// TwinCAT 3 PLC project PLC_HMI
// ProgramVersion: 3.1.4024.0
// libraries:
//   Tc2_DataExchange, * (Beckhoff Automation GmbH)
//   Tc2_Standard, * (Beckhoff Automation GmbH)
//   Tc2_System, * (Beckhoff Automation GmbH)
//   Tc2_Utilities, * (Beckhoff Automation GmbH)
//   Tc3_Database, * (Beckhoff Automation GmbH)
//   Tc3_EventLogger, * (Beckhoff Automation GmbH)
//   Tc3_Module, * (Beckhoff Automation GmbH)
// project tree:
//   DUTs/ ST_Alarm.TcDUT, ST_Error_Station_Handling.TcDUT, ST_Error_Description_Handling.TcDUT, ST_For_Screen.TcDUT, ST_For_Screen_New.TcDUT, ST_UserManagment.TcDUT
//   GVLs/ GVL_Error.TcGVL, GVL_Gauge.TcGVL, GVL_Recipe.TcGVL, GVL_USER.TcGVL, GVL_HIS.TcGVL, GVL_USER_UF.TcGVL, GVL_USER_UP.TcGVL
//   NotUsedPOU/ FB_AssignUserParam.TcPOU, F_ParseKeyValue.TcPOU, F_ParseUserString.TcPOU, F_SplitStringLines.TcPOU, P_EvtLog.TcPOU, P_ParseString.TcPOU, P_UserDataManagment.TcPOU
//   / PlcTask.TcTTO
//   POUs/ FB_Persistent.TcPOU, FB_SaveLineToFile.TcPOU, FB_SaveTextToFile.TcPOU, MAIN.TcPOU, P_ADS_ERR.TcPOU, P_ADS_Gauge.TcPOU, P_Error_Handling.TcPOU, P_Gauge_Measures.TcPOU, P_History_New.TcPOU, P_Recipebackup.TcPOU, P_ADS_1.TcPOU, P_History.TcPOU, P_Time.TcPOU, P_UserManagment.TcPOU, P_UserManagment_UP.TcPOU, P_UserManagment_UF.TcPOU
// real-time tasks:
//   TASK MainTask: cycle T#3ms, priority 20, ADS port 350
//   TASK SafetyTask: cycle T#10ms, priority 21, ADS port 351
//   TASK WeightTask: cycle T#1ms, priority 10, ADS port 352
//   TASK plctaskhmi: cycle T#10ms, priority 30, ADS port 353
//   TASK TaskToRefreshEAP: cycle T#8ms, priority 1, ADS port 301
//   TASK PlcTask: cycle T#10ms, priority 23, ADS port 354

CONFIGURATION PLC_HMI
    RESOURCE PLC ON TwinCAT3
        TASK PlcTask(INTERVAL := T#10ms, PRIORITY := 30);
        PROGRAM MAIN WITH PlcTask : MAIN;
    END_RESOURCE
END_CONFIGURATION

// ---- DUTs/ST_Alarm.TcDUT
TYPE ST_Alarm :
STRUCT
	sTekst1				: WSTRING(255);
	sTekst2				: WSTRING(255);
	sTekst3				: WSTRING(255);
	dtUtworzenia		: DT;
	iNumer				: INT;
	historical_alarm	: WSTRING(1000);
END_STRUCT
END_TYPE

// ---- DUTs/ST_Error_Station_Handling.TcDUT
TYPE ST_Error_Station_Handling :
STRUCT
	udiStationInError			:UDINT;
	wsStasionInError				:WSTRING(255);
END_STRUCT
END_TYPE

// ---- DUTs/ST_Error_Description_Handling.TcDUT
TYPE ST_Error_Description_Handling :
STRUCT
	udiStationErrorCode		:UDINT;
	wsStationErrorDescription	:WSTRING(255);	
END_STRUCT
END_TYPE

// ---- DUTs/ST_For_Screen.TcDUT
TYPE ST_For_Screen :
STRUCT
	data				:WSTRING(255);
	alarmy				:WSTRING(1000);
	user				:WSTRING(80);
	bErrorOccure		:BOOL := FALSE;
END_STRUCT
END_TYPE

// ---- DUTs/ST_For_Screen_New.TcDUT
TYPE ST_For_Screen_New :
STRUCT
	data				:WSTRING(255);
	alarmy				:WSTRING(1000);
	alarmy_id			:UDINT;
	stacja				:UDINT;
	user				:WSTRING(80);
	bErrorOccure		:BOOL := FALSE;
END_STRUCT
END_TYPE

// ---- DUTs/ST_UserManagment.TcDUT
TYPE ST_UserManagment :
STRUCT
	userID 				:	INT;			//numer porządkowy użytkownika
	domain				:	STRING(80);
	enabled				:	BOOL;
	userLogin			:	STRING(80);		//login do zalogowania
	userNameSurname 	:	WSTRING(255);	//imię i nazwisko
	userNameSurnameNumber	:UINT;
	password			:	STRING(255);	//hasło kalwiaturowe
	passwordRFID		:	STRING(255);	//hasło rfid
	passwordQR			:	STRING(255);	//hasło qr
	userGroup			:	STRING(80);		//grupa użytkowników
	userGropuNumber		:	UINT;			//numer grupy
	autoLogOff			:	STRING(80);		//czas do wylogowania
	locale				:	STRING(80);		//gdzie zapisujemy
	timeFormatlocale	:	STRING(80);		//format godziny
	timeZone			:	STRING(80);		//strefa czasowa
	signedPassword		:	STRING(80);		//hasło przekazywane do HMI
END_STRUCT
END_TYPE

// ---- GVLs/GVL_Error.TcGVL
{attribute 'qualified_only'}
VAR_GLOBAL PERSISTENT
	udi_Station_In_Error			:UDINT;
	udi_Station_In_Error_Code		:UDINT;
	ws_Stasion_In_Error				:WSTRING;
	ws_Station_Error_Description		:WSTRING(255);
	ws_Station_Error_Description_2	:WSTRING(255);
	A_Error_station	:ARRAY[0..100] OF ST_Error_Station_Handling; 
	A_Error_description	:ARRAY[0..500] OF ST_Error_Description_Handling;
	
	b_empy_error					:BOOL;
	b_new_system					:BOOL;
END_VAR
VAR_GLOBAL
	logowanie_krok: INT;
END_VAR

// ---- GVLs/GVL_Gauge.TcGVL
{attribute 'qualified_only'}
VAR_GLOBAL
	//input
	lr_WeightMass_recipe	:LREAL;
	lr_Dispencer1WeightMeasured	:LREAL;
	lr_Dispencer2WeightMeasured	:LREAL;
	lr_Dispencer3WeightMeasured	:LREAL;
	lr_Dispencer4WeightMeasured	:LREAL;
	lr_Tolerance_Low			:LREAL;
	lr_Tolerance_High			:LREAL;
	lr_weight_measured_1		:LREAL;
	lr_weight_measured_2		:LREAL;
	lr_weight_measured_3		:LREAL;
	lr_weight_measured_4		:LREAL;
	
	lr_mass_value_1				:LREAL;
	lr_mass_value_2				:LREAL;
	lr_mass_value_3				:LREAL;
	lr_mass_value_4				:LREAL;
	
	
	//output
	lr_out_max_weight_value :LREAL;
	lr_out_min_tolerance_low :LREAL;
	lr_out_max_tolerance_high :LREAL;
	
	lr_out_weight_measured_1 :LREAL;
	lr_out_weight_measured_2 :LREAL;
	lr_out_weight_measured_3 :LREAL;
	lr_out_weight_measured_4 :LREAL;
	
	s_actual_weight_1	:STRING;
	s_actual_weight_2	:STRING;	
	s_actual_weight_3	:STRING;
	s_actual_weight_4	:STRING;
	
	s_actual_weight_1_diff	:STRING;
	s_actual_weight_2_diff	:STRING;
	s_actual_weight_3_diff	:STRING;
	s_actual_weight_4_diff	:STRING;

	s_actual_corr_1		:STRING;
	s_actual_corr_2		:STRING;
	s_actual_corr_3		:STRING;
	s_actual_corr_4		:STRING;	
	
	s_actual_dose_1		:STRING;
	s_actual_dose_2		:STRING;
	s_actual_dose_3		:STRING;
	s_actual_dose_4		:STRING;
	
	lr_corr_add_1	:LREAL;
	lr_corr_sub_1	:LREAL;
	lr_corr_add_2	:LREAL;
	lr_corr_sub_2	:LREAL;
	lr_corr_add_3	:LREAL;
	lr_corr_sub_3	:LREAL;
	lr_corr_add_4	:LREAL;
	lr_corr_sub_4	:LREAL;
	
	s_actual_torque_1	:STRING;
	s_actual_torque_2	:STRING;
	s_actual_torque_diff_1		:STRING;
	s_actual_torque_diff_2		:STRING;
	
	s_actual_level_1	:STRING;
	s_actual_level_2	:STRING;
	
	lr_out_torque_low_1		:LREAL;
	lr_out_torque_low_2		:LREAL;
	lr_out_torque_high_1		:LREAL;
	lr_out_torque_high_2		:LREAL;	

	
END_VAR

// ---- GVLs/GVL_Recipe.TcGVL
{attribute 'qualified_only'}
VAR_GLOBAL
	b_recipe_backup	:BOOL;
END_VAR

// ---- GVLs/GVL_USER.TcGVL
{attribute 'qualified_only'}
VAR_GLOBAL PERSISTENT
		// wejścia cyfrowe
	user_array 					: ARRAY[1..100] OF ST_UserManagment;  // Tablica użytkowników
    currentUser 				: INT := 1;  // Indeks bieżącego użytkownika (zaczyna od 1)
    string_of_properties 		: STRING(1000);  // String z HMI z danymi użytkowników
	outside_accept_login		:BOOL;
	outside_login_pool			:STRING(255);  
	new_user_added				:BOOL;		//dodano użytkownika w PLC
	user_eddited				:BOOL; 		//zedytowano użytkownika w PLC
	b_new_users					:BOOL;		//wgranie uzytkowników
	currentUserName 			:WSTRING(255);
	currentUserGroup			:STRING(80);
	currentUserGroupNumber		:UINT;
	actualUserOn_UserName		:STRING(80);
	b_rewrite_main_users		:BOOL:=FALSE;
	
	logout						:BOOL;
	
	user_try_to_log				:BOOL;
	user_accept_to_log_in		:BOOL;
	no_user_found				:BOOL;
	user_succesed_log			:BOOL;
	putted_user_password		:STRING(255);  //pole w które użytkownik wpisuje hasło
	
	new_user					:BOOL;			//inicjalizacja dodawania nowego użytkownika
	new_user_accept				:BOOL;			//akceptacja dodania nowego użytkownika
	newuserNameSurname 			:WSTRING(255);	//imię i nazwisko
	newpassword					:STRING(255);	//hasło
	newpasswordRFID				:STRING(255);	//hasło rfid
	newpasswordQR				:STRING(255);	//hasło qr
	newuserGroup				:STRING(80);		//grupa użytkowników
	newuserGroupNumber			:UINT;
	newautoLogOff				:STRING(80);			//czas do wylogowania
	newlocale					:STRING(80);		//gdzie zapisujemy
	newtimeFormatlocale			:STRING(80);		//format godziny
	newtimeZone					:STRING(80);		//strefa czasowa
	
	edit_user					:BOOL;				//inicjalizacja edycji użytkownika
	edit_user_accept			:BOOL;			//akceptacja edycji użytkownika
	actual_editted_user			:WSTRING(255);	//wybór aktualnie edytowanego użytkownika
	edituserNameSurname 		:WSTRING(255);	//imię i nazwisko
	editpassword				:STRING(255);	//hasło
	editpasswordRFID			:STRING(255);	//hasło rfid
	editpasswordQR				:STRING(255);	//hasło qr
	edituserGroup				:STRING(80);	//grupa użytkowników
	editUserGroupNumber			:UINT;
	editautoLogOff				:STRING(80);	//czas do wylogowania
	edit_user_qr_or_rfid_password	:BOOL;		//edycja kodów rfid lub qr
		
	//wyjścia cyfrowe
	new_user_add_error			:BOOL;
	edit_user_error				:BOOL;
	bwait						:BOOL;
		
	delete_user						:BOOL;
	delete_user_accept				:BOOL;
	delete_user_error				:BOOL;
	choosen_to_delete				:WSTRING(255);
	user_deleted_succes				:BOOL;
	
	password_to_log_in				:STRING(80); //hasło do pola (1 z 5 (adm, opr, ser, tech, mech)
	
	b_rewrite_users_after_issues	:BOOL:=FALSE;
	
	b_user_drop_the_login			:BOOL;
	
	
	i_choosen_language :INT:=1;
END_VAR

// ---- GVLs/GVL_HIS.TcGVL
{attribute 'qualified_only'}
VAR_GLOBAL PERSISTENT
	// wyjścia cyfrowe
	Historical_array 			: ARRAY [1..1000] OF WSTRING(1000);
	ST_Alarmy 					: ARRAY [1..1000] OF st_for_screen;
	ST_Alarmy_ar1 				: ARRAY [0..28] OF st_for_screen;
	ST_Alarmy_New				:ARRAY  [1..1000] OF st_for_screen_new;
	ST_Alarmy_ar2 				: ARRAY [0..28] OF st_for_screen_new;
	user_for_alarms	 			: WSTRING(80);
	bclearhistory				: BOOL;
	s_time_mainscreen			: WSTRING(80);
	b_next_hist_page			:BOOL;
	b_prev_hist_page			:BOOL;
	i_start_index				:INT:=0;
END_VAR

// ---- GVLs/GVL_USER_UF.TcGVL
{attribute 'qualified_only'}
VAR_GLOBAL PERSISTENT
		// wejścia cyfrowe
	user_array 					: ARRAY[1..100] OF ST_UserManagment;  // Tablica użytkowników
    currentUser 				: INT := 1;  // Indeks bieżącego użytkownika (zaczyna od 1)
    string_of_properties 		: STRING(1000);  // String z HMI z danymi użytkowników
	outside_accept_login		:BOOL;
	outside_login_pool			:STRING(255);  
	new_user_added				:BOOL;		//dodano użytkownika w PLC
	user_eddited				:BOOL; 		//zedytowano użytkownika w PLC
	b_new_users					:BOOL;		//wgranie uzytkowników
	currentUserName 			:WSTRING(255);
	currentUserGroup			:STRING(80);
	actualUserOn_UserName		:STRING(80);
	b_rewrite_main_users		:BOOL:=FALSE;
	
	logout						:BOOL;
	
	user_try_to_log				:BOOL;
	user_accept_to_log_in		:BOOL;
	no_user_found				:BOOL;
	user_succesed_log			:BOOL;
	putted_user_password		:STRING(255);  //pole w które użytkownik wpisuje hasło
	
	new_user					:BOOL;			//inicjalizacja dodawania nowego użytkownika
	new_user_accept				:BOOL;			//akceptacja dodania nowego użytkownika
	newuserNameSurname 			:WSTRING(255);	//imię i nazwisko
	newpassword					:STRING(255);	//hasło
	newpasswordRFID				:STRING(255);	//hasło rfid
	newpasswordQR				:STRING(255);	//hasło qr
	newuserGroup				:STRING(80);		//grupa użytkowników
	newautoLogOff				:STRING(80);			//czas do wylogowania
	newlocale					:STRING(80);		//gdzie zapisujemy
	newtimeFormatlocale			:STRING(80);		//format godziny
	newtimeZone					:STRING(80);		//strefa czasowa
	
	edit_user					:BOOL;				//inicjalizacja edycji użytkownika
	edit_user_accept			:BOOL;			//akceptacja edycji użytkownika
	actual_editted_user			:WSTRING(255);	//wybór aktualnie edytowanego użytkownika
	edituserNameSurname 		:WSTRING(255);	//imię i nazwisko
	editpassword				:STRING(255);	//hasło
	editpasswordRFID			:STRING(255);	//hasło rfid
	editpasswordQR				:STRING(255);	//hasło qr
	edituserGroup				:STRING(80);		//grupa użytkowników
	editautoLogOff				:STRING(80);			//czas do wylogowania
	edit_user_qr_or_rfid_password	:BOOL;		//edycja kodów rfid lub qr
		
	//wyjścia cyfrowe
	new_user_add_error			:BOOL;
	edit_user_error				:BOOL;
	bwait						:BOOL;
		
	delete_user						:BOOL;
	delete_user_accept				:BOOL;
	delete_user_error				:BOOL;
	choosen_to_delete				:WSTRING(255);
	user_deleted_succes				:BOOL;
	
	password_to_log_in				:STRING(80); //hasło do pola (1 z 5 (adm, opr, ser, tech, mech)
	
	b_rewrite_users_after_issues	:BOOL:=FALSE;
	
	
END_VAR

// ---- GVLs/GVL_USER_UP.TcGVL
{attribute 'qualified_only'}
VAR_GLOBAL PERSISTENT
		// wejścia cyfrowe
	user_array 					: ARRAY[1..100] OF ST_UserManagment;  // Tablica użytkowników
    currentUser 				: INT := 1;  // Indeks bieżącego użytkownika (zaczyna od 1)
    string_of_properties 		: STRING(1000);  // String z HMI z danymi użytkowników
	outside_accept_login		:BOOL;
	outside_login_pool			:STRING(255);  
	new_user_added				:BOOL;		//dodano użytkownika w PLC
	user_eddited				:BOOL; 		//zedytowano użytkownika w PLC
	b_new_users					:BOOL;		//wgranie uzytkowników
	currentUserName 			:WSTRING(255);
	currentUserGroup			:STRING(80);
	actualUserOn_UserName		:STRING(80);
	b_rewrite_main_users		:BOOL:=FALSE;
	
	logout						:BOOL;
	
	user_try_to_log				:BOOL;
	user_accept_to_log_in		:BOOL;
	no_user_found				:BOOL;
	user_succesed_log			:BOOL;
	putted_user_password		:STRING(255);  //pole w które użytkownik wpisuje hasło
	
	new_user					:BOOL;			//inicjalizacja dodawania nowego użytkownika
	new_user_accept				:BOOL;			//akceptacja dodania nowego użytkownika
	newuserNameSurname 			:WSTRING(255);	//imię i nazwisko
	newpassword					:STRING(255);	//hasło
	newpasswordRFID				:STRING(255);	//hasło rfid
	newpasswordQR				:STRING(255);	//hasło qr
	newuserGroup				:STRING(80);		//grupa użytkowników
	newautoLogOff				:STRING(80);			//czas do wylogowania
	newlocale					:STRING(80);		//gdzie zapisujemy
	newtimeFormatlocale			:STRING(80);		//format godziny
	newtimeZone					:STRING(80);		//strefa czasowa
	
	edit_user					:BOOL;				//inicjalizacja edycji użytkownika
	edit_user_accept			:BOOL;			//akceptacja edycji użytkownika
	actual_editted_user			:WSTRING(255);	//wybór aktualnie edytowanego użytkownika
	edituserNameSurname 		:WSTRING(255);	//imię i nazwisko
	editpassword				:STRING(255);	//hasło
	editpasswordRFID			:STRING(255);	//hasło rfid
	editpasswordQR				:STRING(255);	//hasło qr
	edituserGroup				:STRING(80);		//grupa użytkowników
	editautoLogOff				:STRING(80);			//czas do wylogowania
	edit_user_qr_or_rfid_password	:BOOL;		//edycja kodów rfid lub qr
		
	//wyjścia cyfrowe
	new_user_add_error			:BOOL;
	edit_user_error				:BOOL;
	bwait						:BOOL;
		
	delete_user						:BOOL;
	delete_user_accept				:BOOL;
	delete_user_error				:BOOL;
	choosen_to_delete				:WSTRING(255);
	user_deleted_succes				:BOOL;
	
	password_to_log_in				:STRING(80); //hasło do pola (1 z 5 (adm, opr, ser, tech, mech)
	
	b_rewrite_users_after_issues	:BOOL:=FALSE;
	
	
END_VAR

// ---- POUs/MAIN.TcPOU
PROGRAM MAIN
VAR
		
END_VAR

P_ADS_1();
P_Time();
P_History();
P_History_New();
P_UserManagment();
P_Recipebackup();
P_Gauge_Measures();
P_ADS_Gauge();
P_ADS_Err();
P_Error_Handling();

END_PROGRAM

// ---- POUs/P_ADS_1.TcPOU
PROGRAM P_ADS_1
VAR
	sTextAlarm1				: WSTRING(255);
	sTextAlarm2				: WSTRING(255);
	sTextAlarm3				: WSTRING(255);
	user					: WSTRING(80);
	iNumberAlarm			: INT;
	bTrigger				: BOOL;
	
	fbRead_1: FB_ReadAdsSymByName;
	fbRead_2: FB_ReadAdsSymByName;
	fbRead_3: FB_ReadAdsSymByName;
	fbCyclicReadout: TON;
	fbRead_4: FB_ReadAdsSymByName;
	fbRead_5: FB_ReadAdsSymByName;
	fbLocaltime: FB_LocalSystemTime;

END_VAR

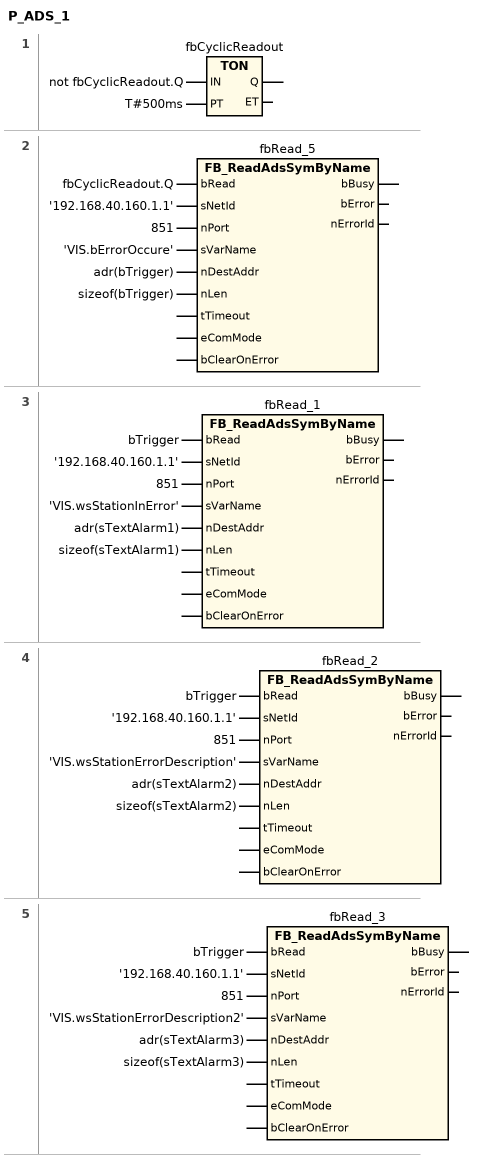
// NETWORK 1
fbCyclicReadout(IN := not fbCyclicReadout.Q, PT := T#500ms); // TON

// NETWORK 2
fbRead_5(
    bRead := fbCyclicReadout.Q,
    sNetId := '192.168.40.160.1.1',
    nPort := 851,
    sVarName := 'VIS.bErrorOccure',
    nDestAddr := adr(bTrigger),
    nLen := sizeof(bTrigger)); // FB_ReadAdsSymByName

// NETWORK 3
fbRead_1(
    bRead := bTrigger,
    sNetId := '192.168.40.160.1.1',
    nPort := 851,
    sVarName := 'VIS.wsStationInError',
    nDestAddr := adr(sTextAlarm1),
    nLen := sizeof(sTextAlarm1)); // FB_ReadAdsSymByName

// NETWORK 4
fbRead_2(
    bRead := bTrigger,
    sNetId := '192.168.40.160.1.1',
    nPort := 851,
    sVarName := 'VIS.wsStationErrorDescription',
    nDestAddr := adr(sTextAlarm2),
    nLen := sizeof(sTextAlarm2)); // FB_ReadAdsSymByName

// NETWORK 5
fbRead_3(
    bRead := bTrigger,
    sNetId := '192.168.40.160.1.1',
    nPort := 851,
    sVarName := 'VIS.wsStationErrorDescription2',
    nDestAddr := adr(sTextAlarm3),
    nLen := sizeof(sTextAlarm3)); // FB_ReadAdsSymByName

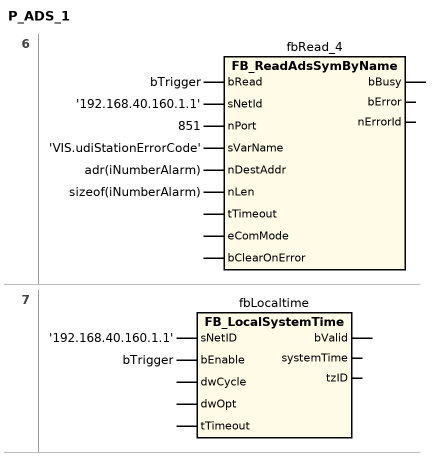
// NETWORK 6
fbRead_4(
    bRead := bTrigger,
    sNetId := '192.168.40.160.1.1',
    nPort := 851,
    sVarName := 'VIS.udiStationErrorCode',
    nDestAddr := adr(iNumberAlarm),
    nLen := sizeof(iNumberAlarm)); // FB_ReadAdsSymByName

// NETWORK 7
fbLocaltime(sNetID := '192.168.40.160.1.1', bEnable := bTrigger); // FB_LocalSystemTime

END_PROGRAM

// ---- POUs/P_Time.TcPOU
PROGRAM P_Time
VAR
    fbSystemTime : GETSYSTEMTIME;
    timeAsFileTime : T_FILETIME;
    timeAsDT : DT;
	actual_date_meawhile :DT;
	s_time_mainscreen	:WSTRING(80);
END_VAR


fbSystemTime(
    timeLoDW => timeAsFileTime.dwLowDateTime,
    timeHiDW => timeAsFileTime.dwHighDateTime 
);
timeAsDT := FILETIME_TO_DT(timeAsFileTime);
actual_date_meawhile:=timeAsDT;
actual_date_meawhile := actual_date_meawhile + T#2H;
s_time_mainscreen := DT_TO_WSTRING(actual_date_meawhile);
s_time_mainscreen := WRIGHT(s_time_mainscreen, WLEN(s_time_mainscreen) - 3);
gvl_his.s_time_mainscreen:=s_time_mainscreen;

END_PROGRAM

// ---- POUs/P_History.TcPOU
PROGRAM P_History
VAR
	nowyAlarm			: BOOL;
	i,j,k,n 			: INT; 
	m					: INT:=0;
	trescAlarmu1		: WSTRING(255);
	trescAlarmu2		: WSTRING(255);
	trescAlarmu3		: WSTRING(255);
	numerAlarmu			: INT;
	aktualnaData		: DT;
	
	bTrigerZapisu 		: R_TRIG;
	
	historical_alarm	: WSTRING(1000);
	tempDateString		: WSTRING(255);
	
	previousTrescAlarmu1 : WSTRING(255);
    previousTrescAlarmu2 : WSTRING(255);
    previousTrescAlarmu3 : WSTRING(255);
    previousNumerAlarmu  : INT;
    previousAktualnaData : DT;
	
	isAlarmChanged : BOOL := FALSE;
	
	isDuplicate: BOOL;
	bCzyszczenie :BOOL :=gvl_his.bclearhistory;
	bDuplikat :	BOOL;
	
	fbPersistent	: FB_Persistent;
	i_start_index		:INT;
	b_next_hist_page_old	:BOOL;
	b_prev_hist_page_old	:BOOL;
END_VAR

fbPersistent(
    bWrite := , 
    tInterval := T#30M, 
    bBusy => , 
    bErr => , 
    udErrID => 
);

trescAlarmu1 := P_ADS_1.sTextAlarm1;
trescAlarmu2 := P_ADS_1.sTextAlarm2;
trescAlarmu3 := P_ADS_1.sTextAlarm3;
numerAlarmu := P_ADS_1.iNumberAlarm;
aktualnaData := P_time.timeAsDT;

isAlarmChanged := (previousTrescAlarmu1 <> trescAlarmu1) OR
                  (previousTrescAlarmu2 <> trescAlarmu2) OR
                  (previousTrescAlarmu3 <> trescAlarmu3) OR
                  (previousNumerAlarmu <> numerAlarmu);

bTrigerZapisu(CLK := P_ADS_1.bTrigger);

IF bTrigerZapisu.Q OR isAlarmChanged THEN
    // Przesuwanie alarmów
    FOR i := 1000 TO 2 BY -1 DO
        GVL_HIS.Historical_array[i] := GVL_HIS.Historical_array[i - 1];
//		GVL_HIS.ST_Alarmy[i] := GVL_HIS.ST_Alarmy[i - 1];
     	GVL_HIS.ST_Alarmy[i].alarmy := GVL_HIS.ST_Alarmy[i - 1].alarmy;  // Przesunięcie struktury do przodu
		GVL_HIS.ST_Alarmy[i].data := GVL_HIS.ST_Alarmy[i - 1].data;
		GVL_HIS.ST_Alarmy[i].user := GVL_HIS.ST_Alarmy[i - 1].user;
		GVL_HIS.ST_Alarmy[i].bErrorOccure := GVL_HIS.ST_Alarmy[i - 1].bErrorOccure;
    END_FOR
    historical_alarm := WCONCAT(UDINT_TO_WSTRING(numerAlarmu), " | ");
    historical_alarm := WCONCAT(historical_alarm, trescAlarmu1);
    historical_alarm := WCONCAT(historical_alarm, " | ");
    historical_alarm := WCONCAT(historical_alarm, trescAlarmu2);
    historical_alarm := WCONCAT(historical_alarm, " | ");
    historical_alarm := WCONCAT(historical_alarm, trescAlarmu3);
    historical_alarm := WCONCAT(historical_alarm, " ");
    aktualnaData := aktualnaData + T#1H;
    tempDateString := DT_TO_WSTRING(aktualnaData);
    tempDateString := WRIGHT(tempDateString, WLEN(tempDateString) - 3);
//	historical_alarm := CONCAT(historical_alarm,tempDateString);

    IF WLEN(historical_alarm) >= 30 THEN
		
        GVL_HIS.Historical_array[1] := historical_alarm;     
		GVL_HIS.ST_Alarmy[1].alarmy := historical_alarm;      
        GVL_HIS.ST_Alarmy[1].data := tempDateString;         
        GVL_HIS.ST_Alarmy[1].user := gvl_his.user_for_alarms;         
        GVL_HIS.ST_Alarmy[1].bErrorOccure := TRUE;
        
        j := 1;
	
        FOR i := 1 TO 1000 DO
            IF WLEN(GVL_HIS.Historical_array[i]) >= 30 THEN
                GVL_HIS.Historical_array[j] := GVL_HIS.Historical_array[i];
				GVL_HIS.ST_Alarmy[j].alarmy := GVL_HIS.ST_Alarmy[i].alarmy; 
				GVL_HIS.ST_Alarmy[j].data := GVL_HIS.ST_Alarmy[i].data;
				GVL_HIS.ST_Alarmy[j].user := GVL_HIS.ST_Alarmy[i].user;
				GVL_HIS.ST_Alarmy[i].bErrorOccure := GVL_HIS.ST_Alarmy[i].bErrorOccure;
                j := j + 1;
            END_IF
        END_FOR

		IF j >= 500 THEN
            FOR i := 500 TO 1000 DO
                GVL_HIS.Historical_array[i] := "";  // Czyszczenie najstarszych wpisów
                GVL_HIS.ST_Alarmy[i].alarmy := "";  // Czyszczenie najstarszych alarmów
                GVL_HIS.ST_Alarmy[i].data := "";  
                GVL_HIS.ST_Alarmy[i].user := "";  
                GVL_HIS.ST_Alarmy[i].bErrorOccure := FALSE;
            END_FOR
            j := 500;  // Aktualizacja j, aby tablica miała maksymalnie 850 alarmów
        END_IF		

        FOR i := j TO 1000 DO
            GVL_HIS.Historical_array[i] := "";
			GVL_HIS.ST_Alarmy[i].alarmy := "";     
       		GVL_HIS.ST_Alarmy[i].data := "";           
      		GVL_HIS.ST_Alarmy[i].user := "";           
      		GVL_HIS.ST_Alarmy[i].bErrorOccure := FALSE;              
        END_FOR		
    END_IF
    
    previousTrescAlarmu1 := trescAlarmu1;
    previousTrescAlarmu2 := trescAlarmu2;
    previousTrescAlarmu3 := trescAlarmu3;
    previousNumerAlarmu := numerAlarmu;
	
	FOR i := 1000 TO 2 BY -1 DO
    isDuplicate := (GVL_HIS.ST_Alarmy[i].alarmy = GVL_HIS.ST_Alarmy[i-1].alarmy) AND
                   (GVL_HIS.ST_Alarmy[i].data = GVL_HIS.ST_Alarmy[i-1].data) AND
                   (GVL_HIS.ST_Alarmy[i].user = GVL_HIS.ST_Alarmy[i-1].user);
    	IF isDuplicate AND bDuplikat THEN
        		FOR j := i TO 1000 - 1 DO
            		GVL_HIS.ST_Alarmy[j] := GVL_HIS.ST_Alarmy[j + 1];
        		END_FOR
        	GVL_HIS.ST_Alarmy[1000].alarmy := "";
        	GVL_HIS.ST_Alarmy[1000].data := "";
        	GVL_HIS.ST_Alarmy[1000].user := "";
    	END_IF
	END_FOR

	IF bCzyszczenie THEN
		FOR i := 1 TO 1000 DO
    		GVL_HIS.ST_Alarmy[i].alarmy := ""; 
    		GVL_HIS.ST_Alarmy[i].data := "";   
    		GVL_HIS.ST_Alarmy[i].user := "";
			GVL_HIS.ST_Alarmy[i].bErrorOccure:=FALSE;    
		END_FOR
	END_IF
END_IF

IF gvl_his.b_next_hist_page = TRUE AND b_next_hist_page_old = FALSE AND gvl_his.i_start_index<20 THEN
	gvl_his.i_start_index:=gvl_his.i_start_index+1;
END_IF

IF gvl_his.b_prev_hist_page = TRUE AND b_prev_hist_page_old = FALSE AND gvl_his.i_start_index>0 THEN
	gvl_his.i_start_index:=gvl_his.i_start_index-1;
END_IF

b_next_hist_page_old := gvl_his.b_next_hist_page;
b_prev_hist_page_old := gvl_his.b_prev_hist_page;

i_start_index := gvl_his.i_start_index * 28;


IF (i_start_index > 0) AND (i_start_index<580) THEN
FOR m := 0 TO 28 DO
        gvl_his.ST_Alarmy_ar1[m].alarmy := gvl_his.ST_Alarmy[i_start_index + m].alarmy;
        gvl_his.ST_Alarmy_ar1[m].bErrorOccure := gvl_his.ST_Alarmy[i_start_index + m].bErrorOccure;
        gvl_his.ST_Alarmy_ar1[m].data := gvl_his.ST_Alarmy[i_start_index + m].data;
        gvl_his.ST_Alarmy_ar1[m].user := gvl_his.ST_Alarmy[i_start_index + m].user;
    END_FOR;
END_IF
IF i_start_index=0 THEN
		FOR m := 1 TO 28 DO
        gvl_his.ST_Alarmy_ar1[m].alarmy := gvl_his.ST_Alarmy[i_start_index + m].alarmy;
        gvl_his.ST_Alarmy_ar1[m].bErrorOccure := gvl_his.ST_Alarmy[i_start_index + m].bErrorOccure;
        gvl_his.ST_Alarmy_ar1[m].data := gvl_his.ST_Alarmy[i_start_index + m].data;
        gvl_his.ST_Alarmy_ar1[m].user := gvl_his.ST_Alarmy[i_start_index + m].user;
    	END_FOR;
END_IF;

END_PROGRAM

// ---- POUs/FB_Persistent.TcPOU
FUNCTION_BLOCK FB_Persistent

(********************************************************************************************************)
(*								Beckhoff Automation Poland												*)
(* 									FB_Persistent 	v1.5												*)
(* 										20.08.2014														*)
(* 							v1.5 - zmiana minimalnego interwalu zapisu									*)
(* 					Blok funkcyjny zapisujący zmienne typu persistent na karcie CF						*)
(* 						Możliwy zapis na żądanie lub z określoną częstotliwością.  						*)
(* 				Pozostawienie wejscia tInterval bez zmiennej wyłacza funkcję zapisu cyklicznego			*)
(* 							Minimalny czas między zapisem cyklicznym 30s								*)
(* 				Konieczne jest dodanie biblioteki TcUtilities.lib, TcSystem.lib oraz TcBase.lib			*)
(*			 UWAGA: Blok przygotowany dla RunTime 1 port 851 - typowa konfiguracja 						*)
(*______________________________________________________________________________________________________*)

VAR_INPUT
	bWrite					: BOOL;						(*Zapis na rozkaz *)
	tInterval				: TIME:=T#71582M47S295MS;	(*Czestotliwosc zapisu na karte CF*)
END_VAR
VAR_OUTPUT
	bBusy					: BOOL;
	bErr					: BOOL;
	udErrID					: UDINT;
END_VAR
VAR
	fbWritePersistentData	: FB_WritePersistentData; 	(* Blok zapisu *)
	t1						: TON;						(* Timer zapisu *)
	_GETCURTASKINDEX		: GETCURTASKINDEX;			(* Informacja o Tasku *)
	BIndex					: BYTE;						(* Nr tasku *)
END_VAR

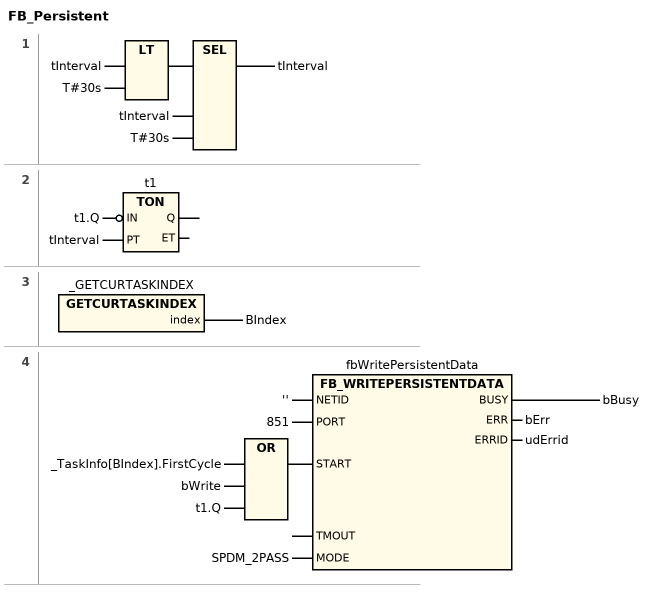
// NETWORK 1
tInterval := SEL(tInterval < T#30s, tInterval, T#30s);

// NETWORK 2
t1(IN := NOT t1.Q, PT := tInterval); // TON

// NETWORK 3
_GETCURTASKINDEX(); // GETCURTASKINDEX
BIndex := _GETCURTASKINDEX.index;

// NETWORK 4
fbWritePersistentData(
    NETID := '',
    PORT := 851,
    START := _TaskInfo[BIndex].FirstCycle OR bWrite OR t1.Q,
    MODE := SPDM_2PASS,
    ERR => bErr,
    ERRID => udErrid); // FB_WRITEPERSISTENTDATA
bBusy := fbWritePersistentData.BUSY;

END_FUNCTION_BLOCK

// ---- POUs/P_History_New.TcPOU
PROGRAM P_History_New
VAR
	nowyAlarm			: BOOL;
	i,j,k,n 			: INT; 
	m					: INT:=0;
	trescAlarmu1		: WSTRING(255);
	trescAlarmu2		: WSTRING(255);
	trescAlarmu3		: WSTRING(255);
	numerAlarmu			: INT;
	aktualnaData		: DT;
	station_id			:UDINT;
	alarm_id			:UDINT;
	
	bTrigerZapisu 		: R_TRIG;
	
	historical_alarm	: WSTRING(1000);
	historical_alarm_id	: UDINT;
	historical_station_id	:UDINT;
	tempDateString		: WSTRING(255);
	
	previousTrescAlarmu1 : WSTRING(255);
    previousTrescAlarmu2 : WSTRING(255);
    previousTrescAlarmu3 : WSTRING(255);
    previousNumerAlarmu  : INT;
    previousAktualnaData : DT;
	
	isAlarmChanged : BOOL := FALSE;
	
	isDuplicate: BOOL;
	bCzyszczenie :BOOL :=gvl_his.bclearhistory;
	bDuplikat :	BOOL;
	
	fbPersistent	: FB_Persistent;
	i_start_index		:INT;
	b_next_hist_page_old	:BOOL;
	b_prev_hist_page_old	:BOOL;
END_VAR

fbPersistent(
    bWrite := , 
    tInterval := T#30M, 
    bBusy => , 
    bErr => , 
    udErrID => 
);

trescAlarmu1 := P_ADS_1.sTextAlarm1;
trescAlarmu2 := P_ADS_1.sTextAlarm2;
trescAlarmu3 := P_ADS_1.sTextAlarm3;
numerAlarmu := P_ADS_1.iNumberAlarm;
aktualnaData := P_time.timeAsDT;
station_id	:=p_ads_err.udiStationInError;
alarm_id	:=p_ads_err.udiStationErrorCode;


isAlarmChanged := (previousTrescAlarmu1 <> trescAlarmu1) OR
                  (previousTrescAlarmu2 <> trescAlarmu2) OR
                  (previousTrescAlarmu3 <> trescAlarmu3) OR
                  (previousNumerAlarmu <> numerAlarmu);

bTrigerZapisu(CLK := P_ADS_1.bTrigger);

IF bTrigerZapisu.Q OR isAlarmChanged THEN
    // Przesuwanie alarmów
    FOR i := 1000 TO 2 BY -1 DO
        GVL_HIS.Historical_array[i] := GVL_HIS.Historical_array[i - 1];
//		GVL_HIS.ST_Alarmy[i] := GVL_HIS.ST_Alarmy[i - 1];
     	GVL_HIS.ST_Alarmy_New[i].alarmy := GVL_HIS.ST_Alarmy_New[i - 1].alarmy;  // Przesunięcie struktury do przodu
		GVL_HIS.ST_Alarmy_New[i].data := GVL_HIS.ST_Alarmy_New[i - 1].data;
		GVL_HIS.ST_Alarmy_New[i].user := GVL_HIS.ST_Alarmy_New[i - 1].user;
		GVL_HIS.ST_Alarmy_New[i].bErrorOccure := GVL_HIS.ST_Alarmy_New[i - 1].bErrorOccure;
		gvl_his.ST_Alarmy_New[i].alarmy_id:=gvl_his.ST_Alarmy_New[i-1].alarmy_id;
		gvl_his.ST_Alarmy_New[i].stacja:=gvl_his.ST_Alarmy_New[i-1].stacja;
    END_FOR
    historical_alarm := WCONCAT(UDINT_TO_WSTRING(numerAlarmu), " | ");
    historical_alarm := WCONCAT(historical_alarm, trescAlarmu1);
    historical_alarm := WCONCAT(historical_alarm, " | ");
    historical_alarm := WCONCAT(historical_alarm, trescAlarmu2);
    historical_alarm := WCONCAT(historical_alarm, " | ");
    historical_alarm := WCONCAT(historical_alarm, trescAlarmu3);
    historical_alarm := WCONCAT(historical_alarm, " ");
    aktualnaData := aktualnaData + T#1H;
    tempDateString := DT_TO_WSTRING(aktualnaData);
    tempDateString := WRIGHT(tempDateString, WLEN(tempDateString) - 3);
	historical_alarm_id:=alarm_id;
	historical_station_id:=station_id;
	
	
	
//	historical_alarm := CONCAT(historical_alarm,tempDateString);

    IF WLEN(historical_alarm) >= 30 THEN
		
        GVL_HIS.Historical_array[1] := historical_alarm;     
		GVL_HIS.ST_Alarmy_new[1].alarmy := historical_alarm;      
        GVL_HIS.ST_Alarmy_new[1].data := tempDateString;         
        GVL_HIS.ST_Alarmy_new[1].user := gvl_his.user_for_alarms;
		GVL_HIS.ST_Alarmy_new[1].alarmy_id:=historical_alarm_id;
		GVL_HIS.ST_Alarmy_new[1].stacja:=historical_station_id;         
        GVL_HIS.ST_Alarmy_new[1].bErrorOccure := TRUE;
        
        j := 1;
	
        FOR i := 1 TO 1000 DO
            IF WLEN(GVL_HIS.Historical_array[i]) >= 30 THEN
                GVL_HIS.Historical_array[j] := GVL_HIS.Historical_array[i];
				GVL_HIS.ST_Alarmy_new[j].alarmy := GVL_HIS.ST_Alarmy_new[i].alarmy; 
				GVL_HIS.ST_Alarmy_new[j].data := GVL_HIS.ST_Alarmy_new[i].data;
				GVL_HIS.ST_Alarmy_new[j].user := GVL_HIS.ST_Alarmy_new[i].user;
				GVL_HIS.ST_Alarmy_new[j].alarmy_id:=GVL_HIS.ST_Alarmy_new[i].alarmy_id;
				GVL_HIS.ST_Alarmy_new[j].stacja:=GVL_HIS.ST_Alarmy_new[i].stacja; 
				GVL_HIS.ST_Alarmy_new[j].bErrorOccure := GVL_HIS.ST_Alarmy_new[i].bErrorOccure;
                j := j + 1;
            END_IF
        END_FOR

		IF j >= 500 THEN
            FOR i := 500 TO 1000 DO
                GVL_HIS.Historical_array[i] := "";  // Czyszczenie najstarszych wpisów
                GVL_HIS.ST_Alarmy_new[i].alarmy := "";  // Czyszczenie najstarszych alarmów
                GVL_HIS.ST_Alarmy_new[i].data := "";  
                GVL_HIS.ST_Alarmy_new[i].user := "";
				GVL_HIS.ST_Alarmy_new[i].alarmy_id:=0;
				GVL_HIS.ST_Alarmy_new[i].stacja:=0;  
                GVL_HIS.ST_Alarmy_new[i].bErrorOccure := FALSE;
            END_FOR
            j := 500;  // Aktualizacja j, aby tablica miała maksymalnie 850 alarmów
        END_IF		

        FOR i := j TO 1000 DO
            GVL_HIS.Historical_array[i] := "";
			GVL_HIS.ST_Alarmy_new[i].alarmy := "";     
       		GVL_HIS.ST_Alarmy_new[i].data := "";           
      		GVL_HIS.ST_Alarmy_new[i].user := "";           
      		GVL_HIS.ST_Alarmy_new[i].bErrorOccure := FALSE;
			GVL_HIS.ST_Alarmy_new[i].alarmy_id:=0;
			GVL_HIS.ST_Alarmy_new[i].stacja:=0;               
        END_FOR		
    END_IF
    
    previousTrescAlarmu1 := trescAlarmu1;
    previousTrescAlarmu2 := trescAlarmu2;
    previousTrescAlarmu3 := trescAlarmu3;
    previousNumerAlarmu := numerAlarmu;
	
	FOR i := 1000 TO 2 BY -1 DO
    isDuplicate := (GVL_HIS.ST_Alarmy_new[i].alarmy = GVL_HIS.ST_Alarmy_new[i-1].alarmy) AND
                   (GVL_HIS.ST_Alarmy_new[i].data = GVL_HIS.ST_Alarmy_new[i-1].data) AND
                   (GVL_HIS.ST_Alarmy_new[i].user = GVL_HIS.ST_Alarmy_new[i-1].user);
    	IF isDuplicate AND bDuplikat THEN
        		FOR j := i TO 1000 - 1 DO
            		GVL_HIS.ST_Alarmy_new[j] := GVL_HIS.ST_Alarmy_new[j + 1];
        		END_FOR
        	GVL_HIS.ST_Alarmy_new[1000].alarmy := "";
        	GVL_HIS.ST_Alarmy_new[1000].data := "";
        	GVL_HIS.ST_Alarmy_new[1000].user := "";
			GVL_HIS.ST_Alarmy_new[1000].alarmy_id:=0;
			GVL_HIS.ST_Alarmy_new[1000].stacja:=0;   
    	END_IF
	END_FOR

	IF bCzyszczenie THEN
		FOR i := 1 TO 1000 DO
    		GVL_HIS.ST_Alarmy_new[i].alarmy := ""; 
    		GVL_HIS.ST_Alarmy_new[i].data := "";   
    		GVL_HIS.ST_Alarmy_new[i].user := "";
			GVL_HIS.ST_Alarmy_new[i].bErrorOccure:=FALSE;
			GVL_HIS.ST_Alarmy_new[i].alarmy_id:=0;
	        GVL_HIS.ST_Alarmy_new[i].stacja:=0;   
		END_FOR
	END_IF
END_IF

IF gvl_his.b_next_hist_page = TRUE AND b_next_hist_page_old = FALSE AND gvl_his.i_start_index<20 THEN
	gvl_his.i_start_index:=gvl_his.i_start_index+1;
END_IF

IF gvl_his.b_prev_hist_page = TRUE AND b_prev_hist_page_old = FALSE AND gvl_his.i_start_index>0 THEN
	gvl_his.i_start_index:=gvl_his.i_start_index-1;
END_IF

b_next_hist_page_old := gvl_his.b_next_hist_page;
b_prev_hist_page_old := gvl_his.b_prev_hist_page;

i_start_index := gvl_his.i_start_index * 28;


IF (i_start_index > 0) AND (i_start_index<580) THEN
FOR m := 0 TO 28 DO
        gvl_his.ST_Alarmy_ar2[m].alarmy := gvl_his.ST_Alarmy_new[i_start_index + m].alarmy;
        gvl_his.ST_Alarmy_ar2[m].bErrorOccure := gvl_his.ST_Alarmy_new[i_start_index + m].bErrorOccure;
        gvl_his.ST_Alarmy_ar2[m].data := gvl_his.ST_Alarmy_new[i_start_index + m].data;
        gvl_his.ST_Alarmy_ar2[m].user := gvl_his.ST_Alarmy_new[i_start_index + m].user;
		gvl_his.ST_Alarmy_ar2[m].stacja := gvl_his.ST_Alarmy_new[i_start_index + m].stacja;
		gvl_his.ST_Alarmy_ar2[m].alarmy_id := gvl_his.ST_Alarmy_new[i_start_index + m].alarmy_id;
		
    END_FOR;
END_IF
IF i_start_index=0 THEN
		FOR m := 1 TO 28 DO
        gvl_his.ST_Alarmy_ar2[m].alarmy := gvl_his.ST_Alarmy_new[i_start_index + m].alarmy;
        gvl_his.ST_Alarmy_ar2[m].bErrorOccure := gvl_his.ST_Alarmy_new[i_start_index + m].bErrorOccure;
        gvl_his.ST_Alarmy_ar2[m].data := gvl_his.ST_Alarmy_new[i_start_index + m].data;
        gvl_his.ST_Alarmy_ar2[m].user := gvl_his.ST_Alarmy_new[i_start_index + m].user;
		gvl_his.ST_Alarmy_ar2[m].stacja := gvl_his.ST_Alarmy_new[i_start_index + m].stacja;
        gvl_his.ST_Alarmy_ar2[m].alarmy_id := gvl_his.ST_Alarmy_new[i_start_index + m].alarmy_id;
    	END_FOR;
END_IF;

END_PROGRAM

// ---- POUs/P_ADS_ERR.TcPOU
PROGRAM P_ADS_ERR
VAR
	udiStationInError				: UDINT;
	udiStationErrorCode				: UDINT;
	sStationErrorDescription2		:WSTRING(255);

	
	fbRead_1: FB_ReadAdsSymByName;
	fbRead_2: FB_ReadAdsSymByName;
	fbRead_3: FB_ReadAdsSymByName;
	fbCyclicReadout: TON;
END_VAR

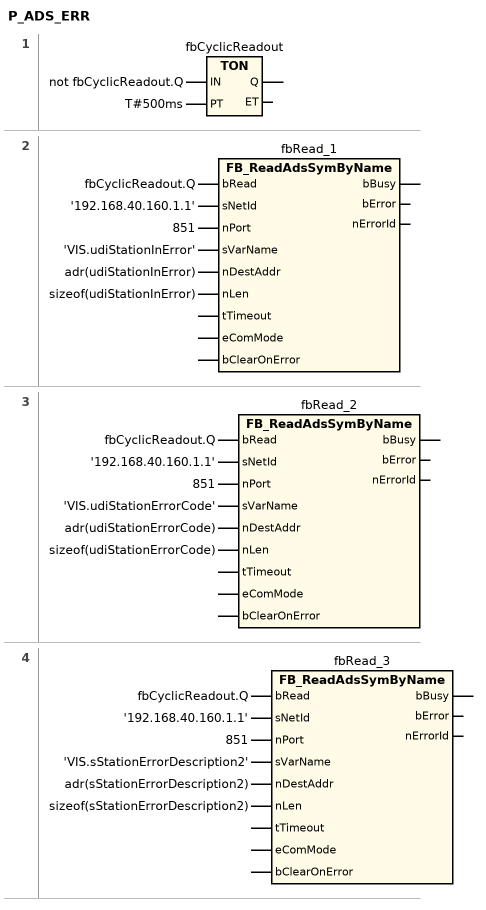
// NETWORK 1
fbCyclicReadout(IN := not fbCyclicReadout.Q, PT := T#500ms); // TON

// NETWORK 2
fbRead_1(
    bRead := fbCyclicReadout.Q,
    sNetId := '192.168.40.160.1.1',
    nPort := 851,
    sVarName := 'VIS.udiStationInError',
    nDestAddr := adr(udiStationInError),
    nLen := sizeof(udiStationInError)); // FB_ReadAdsSymByName

// NETWORK 3
fbRead_2(
    bRead := fbCyclicReadout.Q,
    sNetId := '192.168.40.160.1.1',
    nPort := 851,
    sVarName := 'VIS.udiStationErrorCode',
    nDestAddr := adr(udiStationErrorCode),
    nLen := sizeof(udiStationErrorCode)); // FB_ReadAdsSymByName

// NETWORK 4
fbRead_3(
    bRead := fbCyclicReadout.Q,
    sNetId := '192.168.40.160.1.1',
    nPort := 851,
    sVarName := 'VIS.sStationErrorDescription2',
    nDestAddr := adr(sStationErrorDescription2),
    nLen := sizeof(sStationErrorDescription2)); // FB_ReadAdsSymByName

END_PROGRAM

// ---- POUs/P_UserManagment.TcPOU
PROGRAM P_UserManagment
VAR	
	user_log				:BOOL 				:= GVL_USER.user_try_to_log;           	//użytkownik wywołał okno logowania
	user_accept				:BOOL 				:= GVL_USER.user_accept_to_log_in;     	//użytkownik zaakceptował hasło
	outside_login_accept	:BOOL				:= gvl_user.outside_accept_login;		//przekazanie potwierdzenia procesu logowania
	user_login_error		:BOOL 				:= GVL_USER.no_user_found;				//brak dopasowanego użytkownika
	user_log_succes			:BOOL 				:= GVL_USER.user_succesed_log;			//zalogowano z powodzeniem
	i,j,z					:INT;														//zmienne dla warunków
	bprzypisanie			:BOOL;
	btest					:BOOL:=FALSE;
	k						:INT;
	userExists				:BOOL;														//zmienne dla programu
	outside_login_pool		:STRING(255)		:= gvl_user.outside_login_pool;												//przekazanie loginu do wizualizacji
	user_password			:STRING(255) 		:= GVL_USER.putted_user_password;		//wprowadzone użytkownikiem hasło
	b_new_users				:BOOL;									
	delayTimer: TON;  // Timer do opóźnienia o 500 ms					//nowe wgranie użytkowników
	allowedGroups : ARRAY[1..5] OF STRING(80) := ['Admin', 'Mechanik', 'Operator', 'Technolog', 'Serwis'];
	allowedGroupsNumber	:ARRAY[1..5] OF UINT:=[1,2,3,4,5];
	validGroup    : BOOL;  // Zmienna do walidacji grupy
    uniqueUser    : BOOL;  // Zmienna sprawdzająca unikalność hasła
    freeSlot      : BOOL;  // Zmienna wskazująca wolne miejsce na nowego użytkownika
	bwait	:BOOL :=gvl_user.bwait; //ekran oczekiwania na plc
	bClear	:BOOL:=FALSE;
	iClearArrayNr :INT;
	
	actual_user : WSTRING(255);
	

	new_user				:BOOL := GVL_USER.new_user;			//inicjalizacja dodania nowego użytkownika
	new_user_accept			:BOOL := GVL_USER.new_user_accept;			//akceptacja dodania użytkownika z ekranu
	new_user_added			:BOOL := GVL_USER.new_user_added;			//udane dodanie użytkownika
	new_user_add_error		:BOOL := GVL_USER.new_user_add_error;			//nieudane dodawanie
	newautoLogOff			:STRING(80) := GVL_USER.newautoLogOff;			//czas do wylogowania
	newuserNameSurname 		:WSTRING(255)  := GVL_USER.newuserNameSurname;	//imię i nazwisko				
	newpassword				:STRING(255) := GVL_USER.newpassword;	//hasło
	newpasswordRFID			:STRING(255) := GVL_USER.newpasswordRFID;	//hasło rfid
	newpasswordQR			:STRING(255) := GVL_USER.newpasswordQR;	//hasło qr
	newuserGroup			:STRING(80) := GVL_USER.newuserGroup;		//grupa użytkowników
	newuserLogoffbetween 	:STRING(80);
	
	edit_user						:BOOL := GVL_USER.edit_user;	//inicjalizacja edycji parametrów użytkownika
	edit_user_accept				:BOOL := GVL_USER.edit_user_accept;	//akceptacja wprowadzonych zmiennych z ekranu
	user_eddited					:BOOL := GVL_USER.user_eddited;	//odpowiedź z plc do hmi - udana edycja
	edit_user_qr_or_rfid_password	:BOOL := GVL_USER.edit_user_qr_or_rfid_password;	//edycja rfid lub qr dopisanego do użytkownika
	edit_user_error					:BOOL := GVL_USER.edit_user_error;			//odpowiedź z plc do hmi - nieudana edycja uzytkownika
	editautoLogOff					:STRING(80) := GVL_USER.editautoLogOff;			//czas do wylogowania użytkownika
	edituserNameSurname 			:WSTRING(255) := GVL_USER.edituserNameSurname ;	//imię i nazwisko
	editpassword					:STRING(255) := GVL_USER.editpassword;	//hasło
	editpasswordRFID				:STRING(255) := GVL_USER.editpasswordRFID;	//hasło rfid
	editpasswordQR					:STRING(255) := GVL_USER.editpasswordQR;	//hasło qr
	edituserGroup					:STRING(80) := GVL_USER.edituserGroup;	//grupa użytkowników
	edituserLogoffbetween 	:STRING(80);

	userExists_2			:BOOL;
	userExists_3			:BOOL;
	
	bFirstCycle				:BOOL := FALSE;
	
	iValueForCheck			:INT;
	logowanie_krok	:INT;
END_VAR


bFirstCycle:=TRUE; //Symulacja 1 cyklu sterownika

IF bClear THEN 
    // Sprawdzamy, czy numer wiersza mieści się w zakresie tablicy
    IF (iClearArrayNr >= 1) AND (iClearArrayNr <= 100) THEN
        // Czyszczenie wybranego wiersza tablicy
        GVL_USER.user_array[iClearArrayNr].userID := 0;
        GVL_USER.user_array[iClearArrayNr].domain := '';
        GVL_USER.user_array[iClearArrayNr].enabled := FALSE;
        GVL_USER.user_array[iClearArrayNr].userLogin := '';
        GVL_USER.user_array[iClearArrayNr].userNameSurname := "";  // WSTRING wymaga również pustego ciągu znaków
        GVL_USER.user_array[iClearArrayNr].password := '';
        GVL_USER.user_array[iClearArrayNr].passwordRFID := 'tup';
        GVL_USER.user_array[iClearArrayNr].passwordQR := 'tup';
        GVL_USER.user_array[iClearArrayNr].userGroup := '';
        GVL_USER.user_array[iClearArrayNr].autoLogOff := '';
        GVL_USER.user_array[iClearArrayNr].locale := '';
        GVL_USER.user_array[iClearArrayNr].timeFormatlocale := '';
        GVL_USER.user_array[iClearArrayNr].timeZone := '';
        GVL_USER.user_array[iClearArrayNr].signedPassword := '';
    END_IF

    // Resetowanie flagi bClear po wykonaniu czyszczenia
    bClear := FALSE;
END_IF

// Proces logowania użytkownika GVL_USER.user_try_to_log AND
IF  GVL_USER.user_accept_to_log_in THEN
    GVL_USER.user_succesed_log := FALSE;
    GVL_USER.no_user_found := TRUE;
    gvl_user.bwait := TRUE;
	iValueForCheck:=1;    
	userExists_3 := FALSE;	
    FOR i := 1 TO 100 DO
		
        IF GVL_USER.user_array[i].password = GVL_USER.putted_user_password OR 
           (GVL_USER.user_array[i].passwordRFID = GVL_USER.putted_user_password) OR 
           (GVL_USER.user_array[i].passwordQR = GVL_USER.putted_user_password) THEN
		   
            GVL_USER.currentUser := i;
            userExists_3 := TRUE;
			iValueForCheck:=2;
            EXIT;
			
        END_IF
		
    END_FOR

    IF NOT userExists_3 THEN
		
        GVL_USER.no_user_found := TRUE;
        gvl_user.bwait := FALSE;
		userExists_3 := FALSE;
		iValueForCheck:=3;
		GVL_USER.currentUser := 6;
		gvl_user.currentUserName :="Niezalogowany Użytkownik";
		gvl_user.currentUserGroup :='Niezalogowany';
		gvl_user.currentUserGroupNumber :=0; //
        GVL_USER.user_succesed_log := TRUE;  // Potwierdzenie, że wylogowanie i logowanie zakończyły się sukcesem
        GVL_USER.logout := FALSE;  // Resetowanie sygnału wylogowania
		GVL_USER.putted_user_password:='';
    ELSE

        FOR i := 1 TO 100 DO
            // Sprawdzenie, czy użytkownik jest aktywny
            IF GVL_USER.user_array[i].enabled THEN
                // Sprawdzenie, czy wprowadzone hasło odpowiada loginowi lub RFID/QR
                GVL_USER.no_user_found := FALSE;
				iValueForCheck:=4;
                IF (GVL_USER.user_array[i].password = GVL_USER.putted_user_password) OR
                   (GVL_USER.user_array[i].passwordRFID = GVL_USER.putted_user_password) OR
                   (GVL_USER.user_array[i].passwordQR = GVL_USER.putted_user_password) THEN
                   //delayTimer(IN := TRUE, PT := T#1S);
				   iValueForCheck:=5;
                    // Jeśli wprowadzony kod to RFID lub QR, zastąp go przypisanym hasłem
                    IF GVL_USER.user_array[i].passwordRFID = GVL_USER.putted_user_password THEN
                        GVL_USER.putted_user_password := GVL_USER.user_array[i].password;
						iValueForCheck:=6;
                    	ELSIF GVL_USER.user_array[i].passwordQR = GVL_USER.putted_user_password THEN
                        	GVL_USER.putted_user_password := GVL_USER.user_array[i].password;
							iValueForCheck:=6;
                    END_IF

                 // Sprawdzanie grupy użytkownika i przypisanie odpowiedniej wartości
                 	IF GVL_USER.user_array[i].userGroup = 'Admin' THEN
						iValueForCheck:=7;
                        gvl_user.password_to_log_in := GVL_USER.user_array[i].signedPassword;
                    	ELSIF GVL_USER.user_array[i].userGroup = 'Operator' THEN
                        	gvl_user.password_to_log_in := GVL_USER.user_array[i].signedPassword;
                    	ELSIF GVL_USER.user_array[i].userGroup = 'Serwis' THEN
                        	gvl_user.password_to_log_in := GVL_USER.user_array[i].signedPassword;
                    	ELSIF GVL_USER.user_array[i].userGroup = 'Technolog' THEN
                       		gvl_user.password_to_log_in := GVL_USER.user_array[i].signedPassword;
                    	ELSIF GVL_USER.user_array[i].userGroup = 'Mechanik' THEN
                        	gvl_user.password_to_log_in := GVL_USER.user_array[i].signedPassword;
                    END_IF
                    //IF delayTimer.Q THEN
                		//delayTimer(IN := FALSE);
						iValueForCheck:=8;
						gvl_user.currentUserName := GVL_USER.user_array[i].userNameSurname;
						gvl_user.currentUserGroup := GVL_USER.user_array[i].userGroup;
						gvl_user.currentUserGroupNumber := GVL_USER.user_array[i].userGropuNumber;
                    	GVL_USER.user_succesed_log := TRUE;
                    	GVL_USER.no_user_found := FALSE;                   
                    	gvl_user.bwait := FALSE;
                    	GVL_USER.user_try_to_log := FALSE;
                    	GVL_USER.user_accept_to_log_in := FALSE;
                    // Zerowanie zmiennych po udanym logowaniu
					//gvl_user.outside_accept_login := TRUE;  // Informacja dla wizualizacji
                    //GVL_USER.putted_user_password := '';   // Wyczyszczenie wprowadzonego hasła
                    // Wyczyszczenie hasła do logowania
					//gvl_user.password_to_log_in := '';
					//userExists_3 := FALSE;
					END_IF					
                END_IF
            
        END_FOR
		
        // Jeżeli pętla się zakończy i nie znaleziono użytkownika
        IF NOT GVL_USER.user_succesed_log THEN
            GVL_USER.no_user_found := TRUE; // Ustaw błąd logowania
            gvl_user.bwait := FALSE;
			userExists_3 := FALSE;
			GVL_USER.user_succesed_log := FALSE;
			GVL_USER.putted_user_password:='';
			iValueForCheck:=9;
        END_IF
    END_IF
	GVL_USER.user_succesed_log := FALSE;
	userExists_3:=FALSE;
END_IF
(*IF GVL_USER.user_accept_to_log_in THEN
    logowanie_krok := 1;
END_IF

CASE logowanie_krok OF
    // Krok 0: Stan początkowy
    0:  GVL_USER.no_user_found := FALSE;
        GVL_USER.user_succesed_log := FALSE;
        gvl_user.bwait := FALSE;
        userExists_3 := FALSE;
        iValueForCheck := 0;
    // Krok 1: Inicjalizacja procesu logowania
    1:	logowanie_krok := 2;
        GVL_USER.user_succesed_log := FALSE;
        gvl_user.bwait := TRUE;
        iValueForCheck := 1;
        userExists_3 := FALSE;
    // Krok 2: Szukanie użytkownika na podstawie hasła, RFID lub QR kodu
    2:  FOR i := 1 TO 100 DO
            IF (GVL_USER.user_array[i].password = GVL_USER.putted_user_password) OR 
               (GVL_USER.user_array[i].passwordRFID = GVL_USER.putted_user_password) OR 
               (GVL_USER.user_array[i].passwordQR = GVL_USER.putted_user_password) 
				THEN
                GVL_USER.currentUser := i;
                userExists_3 := TRUE;
				EXIT; // Znaleziono użytkownika, wyjście z pętli
            END_IF
        END_FOR
		
        // Przejdź do kroku 3, jeśli użytkownik nie istnieje
		IF GVL_USER.currentUser <=100 AND GVL_USER.currentUser >0 THEN
        	logowanie_krok := 4;
        		ELSE
            // Jeśli użytkownik istnieje, przejdź do kroku 4
            logowanie_krok := 3;
        	END_IF
    // Krok 3: Obsługa przypadku, gdy użytkownik nie został znaleziony
    3:
        GVL_USER.no_user_found := TRUE;
        gvl_user.bwait := FALSE;
        userExists_3 := FALSE;
        iValueForCheck := 3;
        GVL_USER.putted_user_password := '';
        // Resetowanie zmiennych i powrót do stanu wyjściowego
        logowanie_krok := 0;
    // Krok 4: Sprawdzenie, czy użytkownik jest aktywny
    4:
        IF GVL_USER.user_array[GVL_USER.currentUser].enabled THEN
            GVL_USER.no_user_found := FALSE;
            iValueForCheck := 4;

            // Jeśli wprowadzony kod to RFID lub QR, zastąp go hasłem
            IF GVL_USER.user_array[GVL_USER.currentUser].passwordRFID = GVL_USER.putted_user_password THEN
                GVL_USER.putted_user_password := GVL_USER.user_array[GVL_USER.currentUser].password;
            ELSIF GVL_USER.user_array[GVL_USER.currentUser].passwordQR = GVL_USER.putted_user_password THEN
                GVL_USER.putted_user_password := GVL_USER.user_array[GVL_USER.currentUser].password;
            END_IF

            // Przypisanie hasła w zależności od grupy użytkownika
            CASE GVL_USER.user_array[GVL_USER.currentUser].userGropuNumber OF
                1: gvl_user.password_to_log_in := GVL_USER.user_array[GVL_USER.currentUser].signedPassword;
                2: gvl_user.password_to_log_in := GVL_USER.user_array[GVL_USER.currentUser].signedPassword;
                3: gvl_user.password_to_log_in := GVL_USER.user_array[GVL_USER.currentUser].signedPassword;
                4: gvl_user.password_to_log_in := GVL_USER.user_array[GVL_USER.currentUser].signedPassword;
                5: gvl_user.password_to_log_in := GVL_USER.user_array[GVL_USER.currentUser].signedPassword;
            END_CASE;

            iValueForCheck := 6;

            // Przejdź do kroku 5
            logowanie_krok := 5;
        ELSE
            // Jeżeli użytkownik nie został znaleziony, przejdź do kroku 3
            logowanie_krok := 3;
        END_IF

    // Krok 5: Zakończenie procesu logowania
    5:
        gvl_user.currentUserName := GVL_USER.user_array[GVL_USER.currentUser].userNameSurname;
        gvl_user.currentUserGroup := GVL_USER.user_array[GVL_USER.currentUser].userGroup;
        gvl_user.currentUserGroupNumber := GVL_USER.user_array[GVL_USER.currentUser].userGropuNumber;

        GVL_USER.user_succesed_log := TRUE;
        GVL_USER.no_user_found := FALSE;
        gvl_user.bwait := FALSE;
        GVL_USER.user_try_to_log := FALSE;
        GVL_USER.user_accept_to_log_in := FALSE;

        // Zerowanie zmiennych po udanym logowaniu
        GVL_USER.putted_user_password := '';
        gvl_user.password_to_log_in := '';
        userExists_3 := FALSE;
        iValueForCheck := 7;

        // Resetowanie zmiennych i powrót do stanu wyjściowego
        logowanie_krok := 0;

END_CASE;
*)


// Dodawanie nowego użytkownika
IF GVL_USER.new_user AND GVL_USER.new_user_accept THEN
    GVL_USER.new_user_added := FALSE;
    GVL_USER.new_user_add_error := TRUE;
	gvl_user.bwait := TRUE;
    validGroup := FALSE;  // Na początku zakładamy, że grupa nie jest poprawna
    uniqueUser := TRUE;   // Na początku zakładamy, że hasło jest unikalne
    freeSlot := FALSE;    // Na początku zakładamy, że nie ma wolnego miejsca
    
    // Sprawdzanie, czy wybrana grupa jest jedną z dozwolonych GVL_USER.newuserGroup = allowedGroups[j] 
    FOR j := 1 TO 5 DO
        IF GVL_USER.newuserGroupNumber = allowedGroupsNumber[j]	THEN
            	validGroup := TRUE;  // Jeśli grupa jest dozwolona, ustawiamy na TRUE
        END_IF
    END_FOR

    // Jeśli grupa nie jest poprawna, przerywamy proces dodawania użytkownika
    IF NOT validGroup THEN
        GVL_USER.new_user_add_error := TRUE;
    ELSE
        // Sprawdzanie, czy hasło nie jest już przypisane do innego użytkownika
        FOR i := 7 TO 100 DO
            IF GVL_USER.user_array[i].enabled AND 
               ((GVL_USER.user_array[i].password = GVL_USER.newpassword) OR 
                (GVL_USER.user_array[i].passwordRFID = GVL_USER.newpasswordRFID) OR 
                (GVL_USER.user_array[i].passwordQR = GVL_USER.newpasswordQR)) THEN
                uniqueUser := FALSE;  // Jeśli hasło, RFID lub QR istnieje, ustawiamy na FALSE
            END_IF
        END_FOR

        // Jeśli hasło jest unikalne, szukamy wolnego miejsca w tablicy
        IF uniqueUser THEN
            FOR i := 6 TO 100 DO
                IF NOT GVL_USER.user_array[i].enabled THEN
                    // Przypisanie danych nowego użytkownika
                    GVL_USER.user_array[i].userID := i;
                    GVL_USER.user_array[i].userLogin := GVL_USER.newpassword; // Używamy loginu z hasła
                    GVL_USER.user_array[i].userNameSurname := GVL_USER.newuserNameSurname;
                    GVL_USER.user_array[i].password := GVL_USER.newpassword;

                    // Sprawdzanie, czy pole RFID jest puste - jeśli tak, zapisujemy "tup"
                    IF GVL_USER.newpasswordRFID = '' THEN
                        GVL_USER.user_array[i].passwordRFID := 'tup';
                    ELSE
                        GVL_USER.user_array[i].passwordRFID := GVL_USER.newpasswordRFID;
                    END_IF

                    // Sprawdzanie, czy pole QR jest puste - jeśli tak, zapisujemy "tup"
                    IF GVL_USER.newpasswordQR = '' THEN
                        GVL_USER.user_array[i].passwordQR := 'tup';
                    ELSE
                        GVL_USER.user_array[i].passwordQR := GVL_USER.newpasswordQR;
                    END_IF
                    newuserLogoffbetween:= CONCAT('PT',GVL_USER.newautoLogOff);
                    GVL_USER.user_array[i].userGroup := GVL_USER.newuserGroup;  // Grupa musi być poprawna
                    GVL_USER.user_array[i].autoLogOff := Concat(newuserLogoffbetween,'M');
                    GVL_USER.user_array[i].enabled := TRUE;
					gvl_user.user_array[i].locale:='client';
					gvl_user.user_array[i].timeFormatlocale:='project';
					gvl_user.user_array[i].timeZone:='project';
					gvl_user.user_array[i].domain:='TcHmiUserManagment';
					
					IF GVL_USER.newuserGroupNumber =1 THEN
                        GVL_USER.user_array[i].signedPassword := 'adm';
						GVL_USER.user_array[i].userGropuNumber :=1;
                    ELSIF GVL_USER.newuserGroupNumber =3 THEN
                        GVL_USER.user_array[i].signedPassword := 'opr';
						GVL_USER.user_array[i].userGropuNumber :=3;
                    ELSIF GVL_USER.newuserGroupNumber =5 THEN
                        GVL_USER.user_array[i].signedPassword := 'ser';
						GVL_USER.user_array[i].userGropuNumber :=4;
                    ELSIF GVL_USER.newuserGroupNumber =4 THEN
                        GVL_USER.user_array[i].signedPassword := 'tech';
						GVL_USER.user_array[i].userGropuNumber :=5;
                    ELSIF GVL_USER.newuserGroupNumber =2 THEN
                        GVL_USER.user_array[i].signedPassword := 'mech';
						GVL_USER.user_array[i].userGropuNumber :=2;
                    END_IF
                    
                    // Potwierdzenie dodania nowego użytkownika
                    GVL_USER.new_user_added := TRUE;
                    GVL_USER.new_user_add_error := FALSE;
                    freeSlot := TRUE;  // Znalazło się wolne miejsce
					gvl_user.bwait := FALSE;
                    EXIT;  // Możemy zakończyć pętlę, bo użytkownik został dodany
                END_IF
            END_FOR
        ELSE
            // Hasło, RFID lub QR już istnieje - błąd dodawania użytkownika
            GVL_USER.new_user_add_error := TRUE;
			gvl_user.bwait := FALSE;
        END_IF
    END_IF

    // Jeśli nie znaleziono wolnego miejsca, ustawiamy błąd dodawania
    IF NOT freeSlot THEN
        GVL_USER.new_user_add_error := TRUE;
		gvl_user.bwait := FALSE;
    END_IF
	GVL_USER.new_user:=FALSE;
	validGroup:=FALSE;
	GVL_USER.user_succesed_log := FALSE;
END_IF

IF NOT GVL_USER.new_user THEN
	GVL_USER.new_user_accept:=FALSE;
	gvl_user.bwait := FALSE;
	validGroup:=FALSE;
	GVL_USER.newpasswordQR:='';
	GVL_USER.newpasswordRFID:='';
	newuserLogoffbetween:='';
END_IF



// Edycja istniejącego użytkownika
IF GVL_USER.edit_user AND GVL_USER.edit_user_accept THEN
    GVL_USER.user_eddited := FALSE;
    GVL_USER.edit_user_error := TRUE;
    validGroup := FALSE;  // Na początku zakładamy, że grupa nie jest poprawna
	gvl_user.bwait := TRUE;
    
    // Sprawdzanie, czy użytkownik o podanym imieniu i nazwisku istnieje
    userExists := FALSE;
    FOR i := 1 TO 100 DO
        IF GVL_USER.user_array[i].enabled AND 
           GVL_USER.user_array[i].userNameSurname = GVL_USER.actual_editted_user THEN
            GVL_USER.currentUser := i;
            userExists := TRUE;
            EXIT;  // Zatrzymujemy pętlę, gdy znajdziemy użytkownika
        END_IF
    END_FOR

    // Jeśli użytkownik nie istnieje, kończymy edycję
    IF NOT userExists THEN
        GVL_USER.edit_user_error := TRUE;
        gvl_user.bwait := FALSE;
    ELSE
        // Sprawdzanie, czy użytkownik do edycji jest aktywny
        IF GVL_USER.user_array[GVL_USER.currentUser].enabled THEN
            // Aktualizacja danych użytkownika	

            // Sprawdzanie, czy Imię i Nazwisko ma być zmienione
            IF GVL_USER.edituserNameSurname <> "" THEN
                GVL_USER.user_array[GVL_USER.currentUser].userNameSurname := GVL_USER.edituserNameSurname;
            END_IF
			
            // Sprawdzanie, czy hasło ma być zmienione
			IF GVL_USER.editpassword <> '' THEN
                GVL_USER.user_array[GVL_USER.currentUser].password := GVL_USER.editpassword;
            END_IF

            // Sprawdzanie, czy RFID ma być zmienione
            IF GVL_USER.editpasswordRFID <> '' THEN
                GVL_USER.user_array[GVL_USER.currentUser].passwordRFID := GVL_USER.editpasswordRFID;
            END_IF

            // Sprawdzanie, czy QR ma być zmienione
            IF GVL_USER.editpasswordQR <> '' THEN
                GVL_USER.user_array[GVL_USER.currentUser].passwordQR := GVL_USER.editpasswordQR;
            END_IF
			
			// Sprawdzanie, czy czas wylogowania ma być zmieniony
            IF GVL_USER.editautoLogOff <> '' THEN
				edituserLogoffbetween := CONCAT('PT', GVL_USER.editautoLogOff);
                GVL_USER.user_array[GVL_USER.currentUser].autoLogOff := CONCAT(edituserLogoffbetween, 'M');
            END_IF

            // Sprawdzanie, czy grupa ma być zmieniona
            IF GVL_USER.edituserGroupNumber <> 0 THEN
                // Sprawdzanie, czy wybrana grupa jest jedną z dozwolonych
                FOR j := 1 TO 5 DO
                    IF GVL_USER.edituserGroupNumber = allowedGroupsnumber[j] THEN
                        validGroup := TRUE;  // Jeśli grupa jest dozwolona, ustawiamy na TRUE
                        EXIT;  // Wychodzimy z pętli, bo znaleźliśmy poprawną grupę
                    END_IF
                END_FOR

                // Jeśli grupa nie jest poprawna, przerywamy proces edycji użytkownika
                IF NOT validGroup THEN
                    GVL_USER.edit_user_error := TRUE;
					gvl_user.bwait := FALSE;
					RETURN;  // Kończymy operację, gdy grupa jest nieprawidłowa
                ELSE
                    GVL_USER.user_array[GVL_USER.currentUser].userGroup := GVL_USER.edituserGroup;
                END_IF
            END_IF
            
            // Potwierdzenie edycji użytkownika
            GVL_USER.user_eddited := TRUE;
            GVL_USER.edit_user_error := FALSE;
			gvl_user.bwait := FALSE;
			GVL_USER.user_succesed_log := FALSE;
        END_IF
    END_IF
END_IF

IF NOT GVL_USER.edit_user THEN
	GVL_USER.edit_user_accept:=FALSE;
	gvl_user.bwait := FALSE;
END_IF


// Usuwanie użytkownika
IF GVL_USER.delete_user AND GVL_USER.delete_user_accept THEN
    GVL_USER.delete_user_error := TRUE;  // Zakładamy na początku, że operacja się nie uda
    GVL_USER.user_deleted_succes := FALSE;  // Zmienna sygnalizująca usunięcie użytkownika
    
    // Sprawdzanie, czy użytkownik o podanym imieniu i nazwisku istnieje
    userExists_2 := FALSE;
    FOR i := 1 TO 100 DO
        IF GVL_USER.user_array[i].enabled AND 
           GVL_USER.user_array[i].userNameSurname = GVL_USER.choosen_to_delete THEN
           
            // Użytkownik znaleziony, usuwamy go
            GVL_USER.user_array[i].userID := 0;
            GVL_USER.user_array[i].domain := '';
            GVL_USER.user_array[i].enabled := FALSE;
            GVL_USER.user_array[i].userLogin := '';
            GVL_USER.user_array[i].userNameSurname := "";
            GVL_USER.user_array[i].password := '';
			GVL_USER.user_array[i].signedPassword := '';
            GVL_USER.user_array[i].passwordRFID := '';
            GVL_USER.user_array[i].passwordQR := '';
            GVL_USER.user_array[i].userGroup := '';
			GVL_USER.user_array[i].userGropuNumber:=0;
            GVL_USER.user_array[i].autoLogOff := '';
            GVL_USER.user_array[i].locale := '';
            GVL_USER.user_array[i].timeFormatlocale := '';
            GVL_USER.user_array[i].timeZone := '';
            
            userExists_2 := TRUE;
            GVL_USER.delete_user_error := FALSE;  // Operacja usunięcia powiodła się
            GVL_USER.user_deleted_succes := TRUE;  // Potwierdzenie, że użytkownik został usunięty
            EXIT;  // Zatrzymanie pętli po znalezieniu i usunięciu użytkownika
        END_IF
    END_FOR
    
    // Jeśli użytkownika nie znaleziono, ustaw błąd
    IF NOT userExists_2 THEN
        GVL_USER.delete_user_error := TRUE;  // Nie znaleziono użytkownika
        GVL_USER.user_deleted_succes := FALSE;
    END_IF
	gvl_user.choosen_to_delete:="";
	gvl_user.delete_user_accept:=FALSE;
	userExists_2:=FALSE;
	GVL_USER.user_succesed_log := FALSE;
	GVL_USER.user_deleted_succes := FALSE;
END_IF


// Proces wylogowania użytkownika
IF GVL_USER.logout THEN
    // Czyszczenie danych aktualnie zalogowanego użytkownika
    IF GVL_USER.currentUser >= 1 AND GVL_USER.currentUser <= 100 THEN
       
        // Ustawienie użytkownika "niezalogowany" z wiersza pod indeksem 6
        GVL_USER.currentUser := 6;
		gvl_user.currentUserName :="Niezalogowany Użytkownik";
		gvl_user.currentUserGroup :='Niezalogowany';
		gvl_user.currentUserGroupNumber :=0; //
        GVL_USER.user_succesed_log := TRUE;  // Potwierdzenie, że wylogowanie i logowanie zakończyły się sukcesem
        GVL_USER.logout := FALSE;  // Resetowanie sygnału wylogowania
		GVL_USER.putted_user_password:='';
    END_IF
	GVL_USER.user_succesed_log := FALSE;
END_IF

//Proces nadpisania użytkowników w razie utraty Persistent
IF gvl_user.b_rewrite_users_after_issues OR bFirstCycle 
	THEN
	//admin
	gvl_user.user_array[1].userID:=0;
	gvl_user.user_array[1].enabled:=TRUE;
	gvl_user.user_array[1].userGroup:='Admin';
	gvl_user.user_array[1].userNameSurname:="Administrator";
	gvl_user.user_array[1].password:='adm';
	gvl_user.user_array[1].passwordRFID:='adm';
	gvl_user.user_array[1].passwordQR:='adm';
	gvl_user.user_array[1].userLogin:='adm';
	gvl_user.user_array[1].signedPassword:='adm';
	gvl_user.user_array[1].userGropuNumber:=1;
	//serwis
	gvl_user.user_array[3].userID:=2;
	gvl_user.user_array[3].enabled:=TRUE;
	gvl_user.user_array[3].userGroup:='Serwis';
	gvl_user.user_array[3].userNameSurname:="Serwisant";
	gvl_user.user_array[3].password:='ser';
	gvl_user.user_array[3].passwordRFID:='ser';
	gvl_user.user_array[3].passwordQR:='ser';
	gvl_user.user_array[3].userLogin:='ser';
	gvl_user.user_array[3].signedPassword:='ser';
	gvl_user.user_array[3].userGropuNumber:=4;
	//technolog
	gvl_user.user_array[4].userID:=3;
	gvl_user.user_array[4].enabled:=TRUE;
	gvl_user.user_array[4].userGroup:='Technolog';
	gvl_user.user_array[4].userNameSurname:="Technolog";
	gvl_user.user_array[4].password:='tech';
	gvl_user.user_array[4].passwordRFID:='tech';
	gvl_user.user_array[4].passwordQR:='tech';
	gvl_user.user_array[4].userLogin:='tech';	
	gvl_user.user_array[4].signedPassword:='tech';
	gvl_user.user_array[4].userGropuNumber:=5;
	//operator
	gvl_user.user_array[2].userID:=1;
	gvl_user.user_array[2].enabled:=TRUE;
	gvl_user.user_array[2].userGroup:='Operator';
	gvl_user.user_array[2].userNameSurname:="Operator";
	gvl_user.user_array[2].password:='opr';
	gvl_user.user_array[2].passwordRFID:='opr';
	gvl_user.user_array[2].passwordQR:='opr';
	gvl_user.user_array[2].userLogin:='opr';	
	gvl_user.user_array[2].signedPassword:='opr';
	gvl_user.user_array[2].userGropuNumber:=3;
	//mechanik
	gvl_user.user_array[5].userID:=4;
	gvl_user.user_array[5].enabled:=TRUE;
	gvl_user.user_array[5].userGroup:='Mechanik';
	gvl_user.user_array[5].userNameSurname:="Mechanik";
	gvl_user.user_array[5].password:='mech';
	gvl_user.user_array[5].passwordRFID:='mech';
	gvl_user.user_array[5].passwordQR:='mech';
	gvl_user.user_array[5].userLogin:='mech';	
	gvl_user.user_array[5].signedPassword:='mech';
	gvl_user.user_array[5].userGropuNumber:=2;
	
END_IF

END_PROGRAM

// ---- POUs/P_Recipebackup.TcPOU
PROGRAM P_Recipebackup
VAR
	tonBackup : TON;                     // Timer TON 2 sekund
    tonHour : TON;                       // Timer TON 1 godzina
    bBackupActive : BOOL := FALSE;       // Flaga true
END_VAR

tonHour(IN := NOT tonHour.Q, PT := T#3600S);
IF tonHour.Q THEN
    // Zakończenie liczenia godziny, zaczynamy generowanie sygnału TRUE
    tonHour(IN := FALSE);                // Zresetuj timer godziny
    bBackupActive := TRUE;               // Aktywuj sygnał TRUE
    tonBackup(IN := TRUE, PT := T#2S);   // Zainicjuj timer na 2 sekundy
END_IF

// Timer dla 2 sekundowego sygnału
IF tonBackup.Q THEN
    bBackupActive := FALSE;              // Wyłącz sygnał TRUE po 2 sekundach
    tonBackup(IN := FALSE);              // Zresetuj timer backupu
END_IF
gvl_recipe.b_recipe_backup := bBackupActive;

END_PROGRAM

// ---- POUs/P_Gauge_Measures.TcPOU
PROGRAM P_Gauge_Measures
VAR
	lr_receaved_weight_from_recipe :LREAL;
	lr_max_value :LREAL;
	
	lr_tolerance_actual_low :LREAL;
	lr_tolerance_actual_high :LREAL;
	lr_tolerance_actual_low_weight :LREAL;
	lr_tolerance_actual_high_weight :LREAL;
	
	lr_measured_weight_1 :LREAL;
	s_measured_weight_1_show :STRING;
	s_difference_weight_1_show :STRING;
	lr_difference_weight_1_show_math :LREAL;
	lr_measured_weight_2 :LREAL;
	s_measured_weight_2_show :STRING;
	s_difference_weight_2_show :STRING;
	lr_difference_weight_2_show_math :LREAL;
	lr_measured_weight_3 :LREAL;
	s_measured_weight_3_show :STRING;
	s_difference_weight_3_show :STRING;
	lr_difference_weight_3_show_math :LREAL;
	lr_measured_weight_4 :LREAL;
	s_difference_weight_4_show :STRING;
	s_measured_weight_4_show :STRING;
	lr_difference_weight_4_show_math :LREAL;
	
	s_correction_weight_1	:STRING;
	lr_correction_weight_1_math	:LREAL;
	s_correction_weight_2	:STRING;
	lr_correction_weight_2_math	:LREAL;	
	s_correction_weight_3	:STRING;
	lr_correction_weight_3_math	:LREAL;
	s_correction_weight_4	:STRING;
	lr_correction_weight_4_math	:LREAL;
	
	lr_dosed_1_math			:LREAL;
	s_dosed_1				:STRING;
	lr_dosed_2_math			:LREAL;
	s_dosed_2				:STRING;	
	lr_dosed_3_math			:LREAL;
	s_dosed_3				:STRING;
	lr_dosed_4_math			:LREAL;
	s_dosed_4				:STRING;
	
//korekta	
	lr_add_correction_value_1	:LREAL;
	lr_add_correction_value_2	:LREAL;
	lr_add_correction_value_3	:LREAL;
	lr_add_correction_value_4	:LREAL;
	lr_sub_correction_value_1	:LREAL;
	lr_sub_correction_value_2	:LREAL;
	lr_sub_correction_value_3	:LREAL;
	lr_sub_correction_value_4	:LREAL;	
	
//zakręcanie	
	lr_torque_recipe_set		:LREAL;
	lr_torque_recipe_set_2		:LREAL;
	lr_torque_1					:LREAL;
	s_torque_1					:STRING;
	lr_torque_2					:LREAL;
	s_torque_2					:STRING;
	lr_torq_diff_1				:LREAL;
	lr_torq_diff_2				:LREAL;
	s_torq_diff_1				:STRING;
	s_torq_diff_2				:STRING;
	lr_low_torque_1				:LREAL;
	lr_low_torque_2				:LREAL;
	lr_high_torque_1			:LREAL;
	lr_high_torque_2			:LREAL;
	
//poziomy w zbiornikach
	i_tank_lvl_1				:INT;
	s_tank_lvl_1				:STRING;
	i_tank_lvl_2				:INT;
	s_tank_lvl_2				:STRING;	
	lr_try_value				:lreal;
	
END_VAR

//maksymalny zakres miernika
lr_receaved_weight_from_recipe:=gvl_gauge.lr_WeightMass_recipe; //otrzymanie wartości z receptur
lr_max_value:=2*lr_receaved_weight_from_recipe; //zwiększenie zakresu maksymalnej wagi
gvl_gauge.lr_out_max_weight_value:=lr_max_value; //przepisanie wartości maksymalnej do wykresów wag

//tolerancje dozowników
lr_tolerance_actual_low_weight:=gvl_gauge.lr_Tolerance_Low; //przepisanie wartości z receptury
lr_tolerance_actual_high_weight:=gvl_gauge.lr_Tolerance_High; //przepisanie wartości z receptury
lr_tolerance_actual_low:=lr_receaved_weight_from_recipe-lr_tolerance_actual_low_weight; //ustalenie dolnej granicy
lr_tolerance_actual_high:=lr_receaved_weight_from_recipe+lr_tolerance_actual_high_weight; //ustalenie górnej granicy
//gvl_gauge.lr_out_min_tolerance_low:=lr_tolerance_actual_low*0.775; //przepisanie dolnej granicy
//gvl_gauge.lr_out_max_tolerance_high:=lr_tolerance_actual_high*1.225; //przepisanie górnej granicy 
gvl_gauge.lr_out_min_tolerance_low:=lr_tolerance_actual_low; //przepisanie dolnej granicy
gvl_gauge.lr_out_max_tolerance_high:=lr_tolerance_actual_high; //przepisanie górnej granicy 

//powiększenie wskazania pomiaru
lr_measured_weight_1:=p_ads_gauge.lr_weight_1;
lr_measured_weight_2:=p_ads_gauge.lr_weight_2;
lr_measured_weight_3:=p_ads_gauge.lr_weight_3;
lr_measured_weight_4:=p_ads_gauge.lr_weight_4;

//wskazanie w lewym rogu aktualnej wagi
s_measured_weight_1_show:=CONCAT(LREAL_TO_STRING((TRUNC(p_ads_gauge.lr_weight_1 * 10))/10.0),' g');
s_measured_weight_2_show:=CONCAT(LREAL_TO_STRING((TRUNC(p_ads_gauge.lr_weight_2 * 10))/10.0),' g');
s_measured_weight_3_show:=CONCAT(LREAL_TO_STRING((TRUNC(p_ads_gauge.lr_weight_3 * 10))/10.0),' g');
s_measured_weight_4_show:=CONCAT(LREAL_TO_STRING((TRUNC(p_ads_gauge.lr_weight_4 * 10))/10.0),' g');

gvl_gauge.s_actual_weight_1:=s_measured_weight_1_show;
gvl_gauge.s_actual_weight_2:=s_measured_weight_2_show;
gvl_gauge.s_actual_weight_3:=s_measured_weight_3_show;
gvl_gauge.s_actual_weight_4:=s_measured_weight_4_show;

//wskazanie różnicy pomiaru w prawym rogu
lr_difference_weight_1_show_math:=lr_receaved_weight_from_recipe - p_ads_gauge.lr_weight_1;
s_difference_weight_1_show:=CONCAT((LREAL_TO_FMTSTR(lr_difference_weight_1_show_math,1,TRUE)),' g');

lr_difference_weight_2_show_math:=lr_receaved_weight_from_recipe - p_ads_gauge.lr_weight_2;
s_difference_weight_2_show:=CONCAT((LREAL_TO_FMTSTR(lr_difference_weight_2_show_math,1,TRUE)),' g');

lr_difference_weight_3_show_math:=lr_receaved_weight_from_recipe - p_ads_gauge.lr_weight_3;
s_difference_weight_3_show:=CONCAT((LREAL_TO_FMTSTR(lr_difference_weight_3_show_math,1,TRUE)),' g');

lr_difference_weight_4_show_math:=lr_receaved_weight_from_recipe - p_ads_gauge.lr_weight_4;
s_difference_weight_4_show:=CONCAT((LREAL_TO_FMTSTR(lr_difference_weight_4_show_math,1,TRUE)),' g');

gvl_gauge.s_actual_weight_1_diff:=s_difference_weight_1_show;
gvl_gauge.s_actual_weight_2_diff:=s_difference_weight_2_show;
gvl_gauge.s_actual_weight_3_diff:=s_difference_weight_3_show;
gvl_gauge.s_actual_weight_4_diff:=s_difference_weight_4_show;

//wyświetlanie korekty prawy górny róg
lr_correction_weight_1_math:=p_ads_gauge.lr_correction_weight_1;
s_correction_weight_1:=concat(LREAL_TO_fmtstr(lr_correction_weight_1_math,1,TRUE), ' ml');

lr_correction_weight_2_math:=p_ads_gauge.lr_correction_weight_2;
s_correction_weight_2:=concat(LREAL_TO_fmtstr(lr_correction_weight_2_math,1,TRUE), ' ml');

lr_correction_weight_3_math:=p_ads_gauge.lr_correction_weight_3;
s_correction_weight_3:=concat(LREAL_TO_fmtstr(lr_correction_weight_3_math,1,TRUE), ' ml');

lr_correction_weight_4_math:=p_ads_gauge.lr_correction_weight_4;
s_correction_weight_4:=concat(LREAL_TO_fmtstr(lr_correction_weight_4_math,1,TRUE), ' ml');


gvl_gauge.s_actual_corr_1:=s_correction_weight_1;
gvl_gauge.s_actual_corr_2:=s_correction_weight_2;
gvl_gauge.s_actual_corr_3:=s_correction_weight_3;
gvl_gauge.s_actual_corr_4:=s_correction_weight_4;

//wyświetlanie wydozowanej ilości lewy górny róg
s_dosed_1:=concat(LREAL_TO_fmtstr(p_ads_gauge.lr_dosed_1,1,TRUE),' ml');

s_dosed_2:=concat(LREAL_TO_fmtstr(p_ads_gauge.lr_dosed_2,1,TRUE),' ml');

s_dosed_3:=concat(LREAL_TO_fmtstr(p_ads_gauge.lr_dosed_3,1,TRUE),' ml');

s_dosed_4:=concat(LREAL_TO_fmtstr(p_ads_gauge.lr_dosed_4,1,TRUE),' ml');

gvl_gauge.s_actual_dose_1:=s_dosed_1;
gvl_gauge.s_actual_dose_2:=s_dosed_2;
gvl_gauge.s_actual_dose_3:=s_dosed_3;
gvl_gauge.s_actual_dose_4:=s_dosed_4;

//zmiana korekty dozowania
lr_add_correction_value_1:=lr_correction_weight_1_math+0.5;
lr_add_correction_value_2:=lr_correction_weight_2_math+0.5;
lr_add_correction_value_3:=lr_correction_weight_3_math+0.5;
lr_add_correction_value_4:=lr_correction_weight_4_math+0.5;

lr_sub_correction_value_1:=lr_correction_weight_1_math-0.5;
lr_sub_correction_value_2:=lr_correction_weight_2_math-0.5;
lr_sub_correction_value_3:=lr_correction_weight_3_math-0.5;
lr_sub_correction_value_4:=lr_correction_weight_4_math-0.5;

gvl_gauge.lr_corr_add_1:=lr_add_correction_value_1;
gvl_gauge.lr_corr_add_2:=lr_add_correction_value_2;
gvl_gauge.lr_corr_add_3:=lr_add_correction_value_3;
gvl_gauge.lr_corr_add_4:=lr_add_correction_value_4;
gvl_gauge.lr_corr_sub_1:=lr_sub_correction_value_1;
gvl_gauge.lr_corr_sub_2:=lr_sub_correction_value_2;
gvl_gauge.lr_corr_sub_3:=lr_sub_correction_value_3;
gvl_gauge.lr_corr_sub_4:=lr_sub_correction_value_4;

//momenty i różnice
lr_torque_recipe_set:=p_ads_gauge.lr_screwer_torque_set;
lr_torque_recipe_set_2:=p_ads_gauge.lr_screwer_torque_set_2;
lr_torque_1:=p_ads_gauge.lr_screwer_torque_1;
s_torque_1:=concat(LREAL_TO_fmtstr(lr_torque_1,1,TRUE),' Nm');
gvl_gauge.s_actual_torque_1:=s_torque_1;
lr_torque_2:=p_ads_gauge.lr_screwer_torque_2;
s_torque_2:=concat(LREAL_TO_fmtstr(lr_torque_2,1,TRUE),' Nm');
gvl_gauge.s_actual_torque_2:=s_torque_2;

lr_torq_diff_1:=lr_torque_recipe_set - lr_torque_1;
s_torq_diff_1:=concat(LREAL_TO_FMTSTR(lr_torq_diff_1,1,TRUE),' Nm');
gvl_gauge.s_actual_torque_diff_1:=s_torq_diff_1;
lr_torq_diff_2:=lr_torque_recipe_set_2 - lr_torque_2;
s_torq_diff_2:=concat(LREAL_TO_FMTSTR(lr_torq_diff_2,1,TRUE),' Nm');
gvl_gauge.s_actual_torque_diff_2:=s_torq_diff_2;


gvl_gauge.lr_out_torque_high_1:=lr_torque_recipe_set*1.1;
gvl_gauge.lr_out_torque_high_2:=lr_torque_recipe_set_2*1.1;
gvl_gauge.lr_out_torque_low_1:=lr_torque_recipe_set*0.9;
gvl_gauge.lr_out_torque_low_2:=lr_torque_recipe_set_2*0.9;


//poziomy zbiorników
i_tank_lvl_1:=p_ads_gauge.isensor_value_1;
s_tank_lvl_1:=concat(INT_TO_STRING(i_tank_lvl_1),' mm');
gvl_gauge.s_actual_level_1:=s_tank_lvl_1;
i_tank_lvl_2:=p_ads_gauge.isensor_value_2;
s_tank_lvl_2:=concat(INT_TO_STRING(i_tank_lvl_2),' mm');
gvl_gauge.s_actual_level_2:=s_tank_lvl_2;





(*IF lr_measured_weight_1 > gvl_gauge.lr_out_min_tolerance_low AND lr_measured_weight_1 < gvl_gauge.lr_out_max_tolerance_high
	THEN
	IF lr_measured_weight_1 < lr_receaved_weight_from_recipe AND lr_measured_weight_1>gvl_gauge.lr_out_min_tolerance_low
		THEN			
		gvl_gauge.lr_out_weight_measured_1:=lr_measured_weight_1*1.2;
	ELSIF lr_measured_weight_1 > lr_receaved_weight_from_recipe AND lr_measured_weight_1<gvl_gauge.lr_out_max_tolerance_high
		THEN			
		gvl_gauge.lr_out_weight_measured_1:=lr_measured_weight_1*0.8;		
	END_IF		
END_IF*)

gvl_gauge.lr_out_weight_measured_1:=lr_measured_weight_1;


(*	IF lr_measured_weight_1 < lr_receaved_weight_from_recipe AND lr_measured_weight_1>gvl_gauge.lr_out_min_tolerance_low
		THEN			
		gvl_gauge.lr_out_weight_measured_1:=lr_measured_weight_1*1.225;
	ELSIF lr_measured_weight_1 > lr_receaved_weight_from_recipe AND lr_measured_weight_1<gvl_gauge.lr_out_max_tolerance_high
		THEN			
		gvl_gauge.lr_out_weight_measured_1:=lr_measured_weight_1*0.775;		
	ELSIF lr_measured_weight_1 < lr_receaved_weight_from_recipe AND lr_measured_weight_1<gvl_gauge.lr_out_min_tolerance_low
		THEN 
		gvl_gauge.lr_out_weight_measured_1:=0;
	ELSIF lr_measured_weight_1 > lr_receaved_weight_from_recipe AND lr_measured_weight_1>gvl_gauge.lr_out_max_tolerance_high
		THEN 
		gvl_gauge.lr_out_weight_measured_1:=lr_max_value;	
	END_IF		
*)
(*IF lr_measured_weight_2 > gvl_gauge.lr_out_min_tolerance_low AND lr_measured_weight_2 < gvl_gauge.lr_out_max_tolerance_high
	THEN
	IF lr_measured_weight_2 < lr_receaved_weight_from_recipe AND lr_measured_weight_2>gvl_gauge.lr_out_min_tolerance_low
		THEN			
		gvl_gauge.lr_out_weight_measured_2:=lr_measured_weight_2*1.06;
	ELSIF lr_measured_weight_2 > lr_receaved_weight_from_recipe AND lr_measured_weight_2<gvl_gauge.lr_out_max_tolerance_high
		THEN			
		gvl_gauge.lr_out_weight_measured_2:=lr_measured_weight_2*0.94;		
	END_IF		
END_IF*)

		gvl_gauge.lr_out_weight_measured_2:=lr_measured_weight_2;

(*	IF lr_measured_weight_2 < lr_receaved_weight_from_recipe AND lr_measured_weight_2>gvl_gauge.lr_out_min_tolerance_low
		THEN			
		gvl_gauge.lr_out_weight_measured_2:=lr_measured_weight_2*1.225;
	ELSIF lr_measured_weight_2 > lr_receaved_weight_from_recipe AND lr_measured_weight_2<gvl_gauge.lr_out_max_tolerance_high
		THEN			
		gvl_gauge.lr_out_weight_measured_2:=lr_measured_weight_2*0.775;		
	ELSIF lr_measured_weight_2 < lr_receaved_weight_from_recipe AND lr_measured_weight_2<gvl_gauge.lr_out_min_tolerance_low
		THEN 
		gvl_gauge.lr_out_weight_measured_2:=0;
	ELSIF lr_measured_weight_2 > lr_receaved_weight_from_recipe AND lr_measured_weight_2>gvl_gauge.lr_out_max_tolerance_high
		THEN 
		gvl_gauge.lr_out_weight_measured_2:=lr_max_value;	
	END_IF	
*)
(*IF lr_measured_weight_3 > gvl_gauge.lr_out_min_tolerance_low AND lr_measured_weight_3 < gvl_gauge.lr_out_max_tolerance_high
	THEN
	IF lr_measured_weight_3 < lr_receaved_weight_from_recipe AND lr_measured_weight_3>gvl_gauge.lr_out_min_tolerance_low
		THEN			
		gvl_gauge.lr_out_weight_measured_3:=lr_measured_weight_3*1.06;
	ELSIF lr_measured_weight_3 > lr_receaved_weight_from_recipe AND lr_measured_weight_3<gvl_gauge.lr_out_max_tolerance_high
		THEN			
		gvl_gauge.lr_out_weight_measured_3:=lr_measured_weight_3*0.94;		
	END_IF		
END_IF*)

gvl_gauge.lr_out_weight_measured_3:=lr_measured_weight_3;

(*	IF lr_measured_weight_3 < lr_receaved_weight_from_recipe AND lr_measured_weight_3>gvl_gauge.lr_out_min_tolerance_low
		THEN			
		gvl_gauge.lr_out_weight_measured_3:=lr_measured_weight_3*1.225;
	ELSIF lr_measured_weight_3 > lr_receaved_weight_from_recipe AND lr_measured_weight_3<gvl_gauge.lr_out_max_tolerance_high
		THEN			
		gvl_gauge.lr_out_weight_measured_3:=lr_measured_weight_3*0.775;
	ELSIF lr_measured_weight_3 < lr_receaved_weight_from_recipe AND lr_measured_weight_3<gvl_gauge.lr_out_min_tolerance_low
		THEN 
		gvl_gauge.lr_out_weight_measured_3:=0;
	ELSIF lr_measured_weight_3 > lr_receaved_weight_from_recipe AND lr_measured_weight_3>gvl_gauge.lr_out_max_tolerance_high
		THEN 
		gvl_gauge.lr_out_weight_measured_3:=lr_max_value;			
	END_IF		
*)
(*IF lr_measured_weight_4 > gvl_gauge.lr_out_min_tolerance_low AND lr_measured_weight_4 < gvl_gauge.lr_out_max_tolerance_high
	THEN
	IF lr_measured_weight_4 < lr_receaved_weight_from_recipe AND lr_measured_weight_4>gvl_gauge.lr_out_min_tolerance_low
		THEN			
		gvl_gauge.lr_out_weight_measured_4:=lr_measured_weight_4*1.06;
	ELSIF lr_measured_weight_4 > lr_receaved_weight_from_recipe AND lr_measured_weight_4<gvl_gauge.lr_out_max_tolerance_high
		THEN			
		gvl_gauge.lr_out_weight_measured_4:=lr_measured_weight_4*0.94;		
	END_IF		
END_IF*)

gvl_gauge.lr_out_weight_measured_4:=lr_measured_weight_4;

(*	IF lr_measured_weight_4 < lr_receaved_weight_from_recipe AND lr_measured_weight_4>gvl_gauge.lr_out_min_tolerance_low
		THEN			
		gvl_gauge.lr_out_weight_measured_4:=lr_measured_weight_4*1.225;
	ELSIF lr_measured_weight_4 > lr_receaved_weight_from_recipe AND lr_measured_weight_4<gvl_gauge.lr_out_max_tolerance_high
		THEN			
		gvl_gauge.lr_out_weight_measured_4:=lr_measured_weight_4*0.775;
	ELSIF lr_measured_weight_4 < lr_receaved_weight_from_recipe AND lr_measured_weight_4<gvl_gauge.lr_out_min_tolerance_low
		THEN 
		gvl_gauge.lr_out_weight_measured_4:=0;
	ELSIF lr_measured_weight_4 > lr_receaved_weight_from_recipe AND lr_measured_weight_4>gvl_gauge.lr_out_max_tolerance_high
		THEN 
		gvl_gauge.lr_out_weight_measured_4:=lr_max_value;	
	END_IF	
	*)

END_PROGRAM

// ---- POUs/P_ADS_Gauge.TcPOU
PROGRAM P_ADS_Gauge
VAR
	bTrigger				: BOOL;
	lr_weight_1				:LREAL;
	lr_weight_2				:LREAL;
	lr_weight_3				:LREAL;
	lr_weight_4				:LREAL;
	
	lr_correction_weight_1  :LREAL;
	lr_correction_weight_2  :LREAL;
	lr_correction_weight_3  :LREAL;
	lr_correction_weight_4  :LREAL;	
	
	lr_dosed_1				:LREAL;
	lr_dosed_2				:LREAL;
	lr_dosed_3				:LREAL;
	lr_dosed_4				:LREAL;
	
	isensor_value_1			:INT;
	isensor_value_2			:INT;
	
	lr_screwer_torque_1		:LREAL;
	lr_screwer_torque_2		:LREAL;
	lr_screwer_torque_set	:LREAL;
	lr_screwer_torque_set_2	:LREAL;
//weight measureg
	fbRead_1: FB_ReadAdsSymByName;
	fbRead_2: FB_ReadAdsSymByName;
	fbRead_3: FB_ReadAdsSymByName;
	fbRead_4: FB_ReadAdsSymByName;
//correction weight	
	fbRead_5: FB_ReadAdsSymByName;
	fbRead_6: FB_ReadAdsSymByName;
	fbRead_7: FB_ReadAdsSymByName;
	fbRead_8: FB_ReadAdsSymByName;
//dose volume
	fbRead_9: FB_ReadAdsSymByName;
	fbRead_10: FB_ReadAdsSymByName;
	fbRead_11: FB_ReadAdsSymByName;
	fbRead_12: FB_ReadAdsSymByName;
//tank level
	fbRead_13: FB_ReadAdsSymByName;
	fbRead_14: FB_ReadAdsSymByName;
//Screwer torque
	fbRead_17: FB_ReadAdsSymByName;
	fbRead_16: FB_ReadAdsSymByName;
//Screwer torque recipe
	fbRead_15: FB_ReadAdsSymByName;
	fbRead_18: FB_ReadAdsSymByName;
	
	fbCyclicReadout: TON;
END_VAR

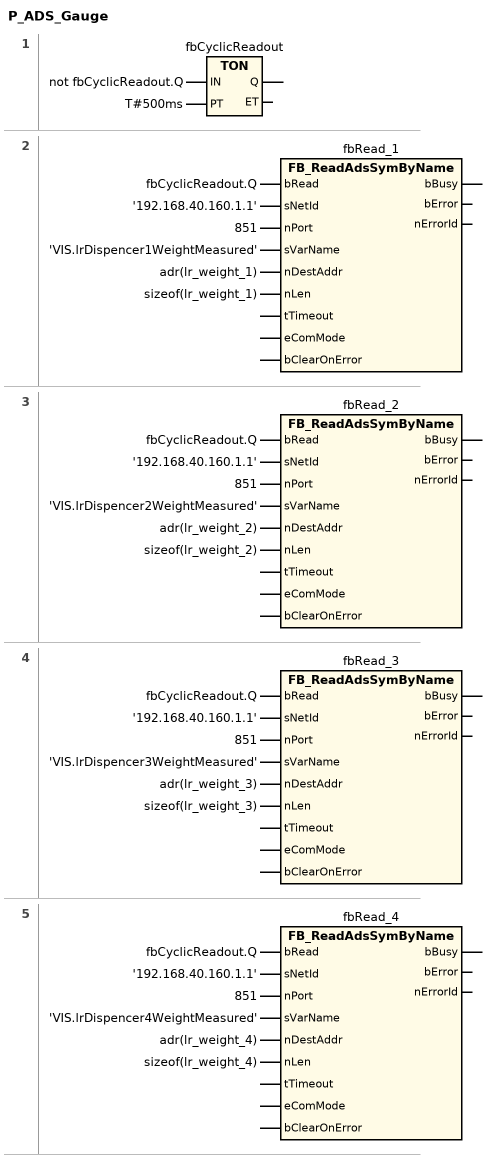
// NETWORK 1
fbCyclicReadout(IN := not fbCyclicReadout.Q, PT := T#500ms); // TON

// NETWORK 2
fbRead_1(
    bRead := fbCyclicReadout.Q,
    sNetId := '192.168.40.160.1.1',
    nPort := 851,
    sVarName := 'VIS.lrDispencer1WeightMeasured',
    nDestAddr := adr(lr_weight_1),
    nLen := sizeof(lr_weight_1)); // FB_ReadAdsSymByName

// NETWORK 3
fbRead_2(
    bRead := fbCyclicReadout.Q,
    sNetId := '192.168.40.160.1.1',
    nPort := 851,
    sVarName := 'VIS.lrDispencer2WeightMeasured',
    nDestAddr := adr(lr_weight_2),
    nLen := sizeof(lr_weight_2)); // FB_ReadAdsSymByName

// NETWORK 4
fbRead_3(
    bRead := fbCyclicReadout.Q,
    sNetId := '192.168.40.160.1.1',
    nPort := 851,
    sVarName := 'VIS.lrDispencer3WeightMeasured',
    nDestAddr := adr(lr_weight_3),
    nLen := sizeof(lr_weight_3)); // FB_ReadAdsSymByName

// NETWORK 5
fbRead_4(
    bRead := fbCyclicReadout.Q,
    sNetId := '192.168.40.160.1.1',
    nPort := 851,
    sVarName := 'VIS.lrDispencer4WeightMeasured',
    nDestAddr := adr(lr_weight_4),
    nLen := sizeof(lr_weight_4)); // FB_ReadAdsSymByName

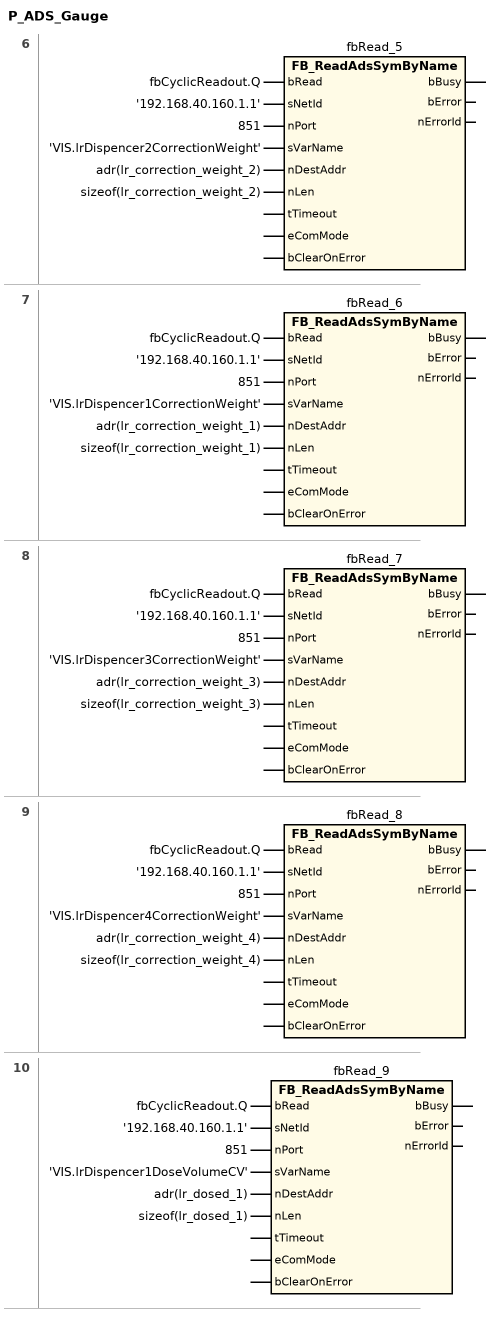
// NETWORK 6
fbRead_5(
    bRead := fbCyclicReadout.Q,
    sNetId := '192.168.40.160.1.1',
    nPort := 851,
    sVarName := 'VIS.lrDispencer2CorrectionWeight',
    nDestAddr := adr(lr_correction_weight_2),
    nLen := sizeof(lr_correction_weight_2)); // FB_ReadAdsSymByName

// NETWORK 7
fbRead_6(
    bRead := fbCyclicReadout.Q,
    sNetId := '192.168.40.160.1.1',
    nPort := 851,
    sVarName := 'VIS.lrDispencer1CorrectionWeight',
    nDestAddr := adr(lr_correction_weight_1),
    nLen := sizeof(lr_correction_weight_1)); // FB_ReadAdsSymByName

// NETWORK 8
fbRead_7(
    bRead := fbCyclicReadout.Q,
    sNetId := '192.168.40.160.1.1',
    nPort := 851,
    sVarName := 'VIS.lrDispencer3CorrectionWeight',
    nDestAddr := adr(lr_correction_weight_3),
    nLen := sizeof(lr_correction_weight_3)); // FB_ReadAdsSymByName

// NETWORK 9
fbRead_8(
    bRead := fbCyclicReadout.Q,
    sNetId := '192.168.40.160.1.1',
    nPort := 851,
    sVarName := 'VIS.lrDispencer4CorrectionWeight',
    nDestAddr := adr(lr_correction_weight_4),
    nLen := sizeof(lr_correction_weight_4)); // FB_ReadAdsSymByName

// NETWORK 10
fbRead_9(
    bRead := fbCyclicReadout.Q,
    sNetId := '192.168.40.160.1.1',
    nPort := 851,
    sVarName := 'VIS.lrDispencer1DoseVolumeCV',
    nDestAddr := adr(lr_dosed_1),
    nLen := sizeof(lr_dosed_1)); // FB_ReadAdsSymByName

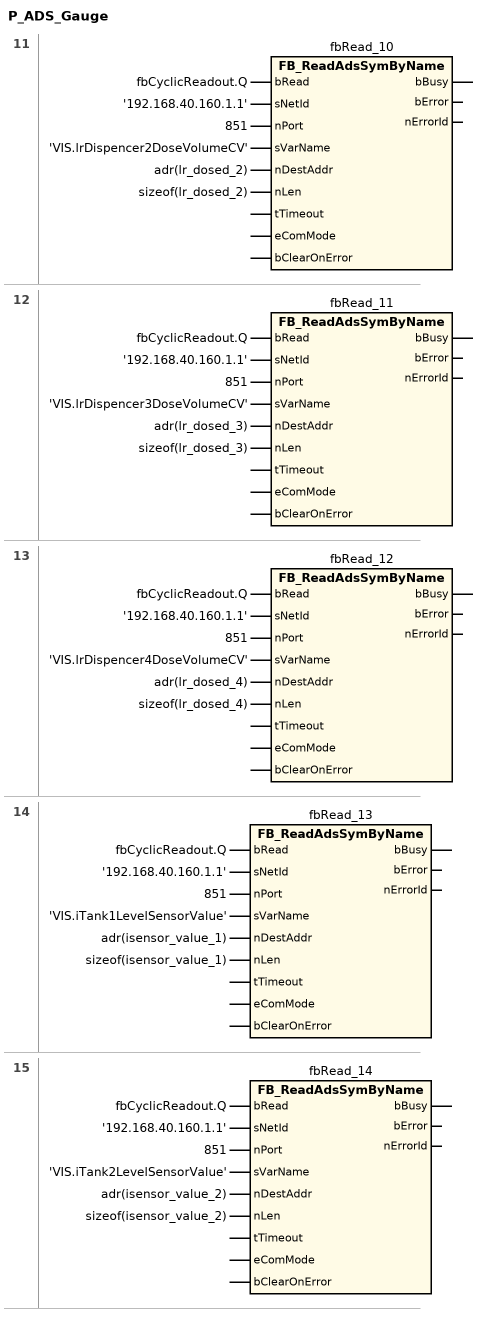
// NETWORK 11
fbRead_10(
    bRead := fbCyclicReadout.Q,
    sNetId := '192.168.40.160.1.1',
    nPort := 851,
    sVarName := 'VIS.lrDispencer2DoseVolumeCV',
    nDestAddr := adr(lr_dosed_2),
    nLen := sizeof(lr_dosed_2)); // FB_ReadAdsSymByName

// NETWORK 12
fbRead_11(
    bRead := fbCyclicReadout.Q,
    sNetId := '192.168.40.160.1.1',
    nPort := 851,
    sVarName := 'VIS.lrDispencer3DoseVolumeCV',
    nDestAddr := adr(lr_dosed_3),
    nLen := sizeof(lr_dosed_3)); // FB_ReadAdsSymByName

// NETWORK 13
fbRead_12(
    bRead := fbCyclicReadout.Q,
    sNetId := '192.168.40.160.1.1',
    nPort := 851,
    sVarName := 'VIS.lrDispencer4DoseVolumeCV',
    nDestAddr := adr(lr_dosed_4),
    nLen := sizeof(lr_dosed_4)); // FB_ReadAdsSymByName

// NETWORK 14
fbRead_13(
    bRead := fbCyclicReadout.Q,
    sNetId := '192.168.40.160.1.1',
    nPort := 851,
    sVarName := 'VIS.iTank1LevelSensorValue',
    nDestAddr := adr(isensor_value_1),
    nLen := sizeof(isensor_value_1)); // FB_ReadAdsSymByName

// NETWORK 15
fbRead_14(
    bRead := fbCyclicReadout.Q,
    sNetId := '192.168.40.160.1.1',
    nPort := 851,
    sVarName := 'VIS.iTank2LevelSensorValue',
    nDestAddr := adr(isensor_value_2),
    nLen := sizeof(isensor_value_2)); // FB_ReadAdsSymByName

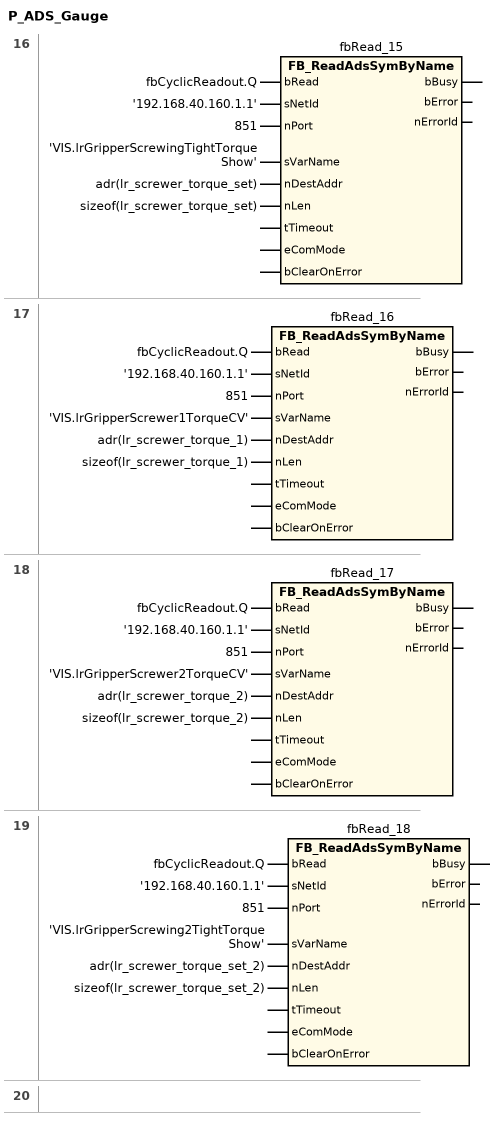
// NETWORK 16
fbRead_15(
    bRead := fbCyclicReadout.Q,
    sNetId := '192.168.40.160.1.1',
    nPort := 851,
    sVarName := 'VIS.lrGripperScrewingTightTorqueShow',
    nDestAddr := adr(lr_screwer_torque_set),
    nLen := sizeof(lr_screwer_torque_set)); // FB_ReadAdsSymByName

// NETWORK 17
fbRead_16(
    bRead := fbCyclicReadout.Q,
    sNetId := '192.168.40.160.1.1',
    nPort := 851,
    sVarName := 'VIS.lrGripperScrewer1TorqueCV',
    nDestAddr := adr(lr_screwer_torque_1),
    nLen := sizeof(lr_screwer_torque_1)); // FB_ReadAdsSymByName

// NETWORK 18
fbRead_17(
    bRead := fbCyclicReadout.Q,
    sNetId := '192.168.40.160.1.1',
    nPort := 851,
    sVarName := 'VIS.lrGripperScrewer2TorqueCV',
    nDestAddr := adr(lr_screwer_torque_2),
    nLen := sizeof(lr_screwer_torque_2)); // FB_ReadAdsSymByName

// NETWORK 19
fbRead_18(
    bRead := fbCyclicReadout.Q,
    sNetId := '192.168.40.160.1.1',
    nPort := 851,
    sVarName := 'VIS.lrGripperScrewing2TightTorqueShow',
    nDestAddr := adr(lr_screwer_torque_set_2),
    nLen := sizeof(lr_screwer_torque_set_2)); // FB_ReadAdsSymByName

// NETWORK 20

END_PROGRAM

// ---- POUs/P_Error_Handling.TcPOU
PROGRAM P_Error_Handling 
VAR
	bErrorOccure	:BOOL;
	bErrorTrig		:R_trig;
	bNewSystem		:BOOL:=TRUE;

	udiStationInError				: UDINT;
	previousStationErrorCode		: UDINT;
	udiStationErrorCode				: UDINT;
	i,j,k,l,n,m: INT;
	bAlarmExist				:BOOL;
	i_current_alarm			:INT;
	j_current_alarm			: INT;
	bAlarmExist_j: BOOL;
	bAlarmExist_i: BOOL;
	b_write:BOOL;
	b_write2:BOOL;
	wstrStation :WSTRING(255);
	wstrStation2 :WSTRING(255);
	bFirstCycle				:BOOL := FALSE;
	values: ARRAY[1..175] OF INT := [
        1, 2, 3, 4, 5, 6, 7, 8, 9, 10, 11, 12, 13, 14, 15, 16, 17, 
        31, 32, 33, 34, 35, 36, 37, 38, 39, 40, 41, 42, 43, 44, 45, 
        46, 47, 48, 49, 50, 51, 52, 53, 54, 55, 56, 57, 58, 59, 60, 
        61, 62, 63, 64, 65, 66, 67, 68, 69, 70, 71, 72, 73, 74, 75, 
        76, 77, 78, 79, 84, 85, 86, 87, 88, 89, 90, 91, 92, 93, 94, 
        95, 96, 97, 98, 99, 101, 102, 103, 104, 105, 106, 107, 111, 
        112, 121, 122, 123, 124, 125, 131, 132, 141, 142, 143, 144, 
        145, 146, 147, 148, 149, 150, 151, 161, 162, 163, 164, 165, 
        171, 172, 173, 174, 175, 181, 182, 191, 192, 193, 194, 195, 
        196, 201, 202, 211, 221, 222, 223, 224, 225, 226, 227, 228, 
        229, 230, 241, 242, 243, 251, 252, 253, 254, 255, 256, 257, 
        258, 261, 262, 263, 264, 265, 266, 271, 272, 273, 281, 282, 
        283, 284, 285, 291, 292, 293, 294, 295, 296, 297, 301, 302, 
        303
    ];

	rTrigError_1:r_trig;
	bisAlarmChanged:BOOL;
END_VAR

bFirstCycle:=TRUE;
bErrorOccure			:= p_ads_1.bTrigger;
bErrorTrig				(CLK:= bErrorOccure);
//udiStationInError		:=P_ADS_ERR.udiStationInError;
IF P_ADS_ERR.udiStationInError=0 THEN
	udiStationInError:=1;
	ELSE
	udiStationInError:= P_ADS_ERR.udiStationInError;
END_IF
udiStationErrorCode:=P_ADS_ERR.udiStationErrorCode;

IF bErrorTrig.Q OR rTrigError_1.Q //AND bNewSystem 
THEN
	bAlarmExist_j:=FALSE;
	bAlarmExist_i:=FALSE;
	FOR i:=1 TO 57 DO
		 IF gvl_error.A_Error_station[i].udiStationInError 		= udiStationInError THEN
            i_current_alarm						:= i;
            bAlarmExist_i 						:= TRUE;
			gvl_error.b_empy_error:=FALSE;
			 EXIT;       
		ELSE
			gvl_error.b_empy_error:=TRUE;
			bAlarmExist_i 						:= FALSE;	
		END_IF		
	END_FOR
		FOR j:=1 TO 177 DO
		 IF gvl_error.A_Error_description[j].udiStationErrorCode 		= udiStationErrorCode THEN
            j_current_alarm						:= j;
            bAlarmExist_j 						:= TRUE;
			gvl_error.b_empy_error:=FALSE;
			previousStationErrorCode:=udiStationErrorCode;
			EXIT;
		ELSE
			gvl_error.b_empy_error:=TRUE;
			bAlarmExist_j 						:=FALSE;
            
        END_IF		
	END_FOR
		
	IF  bAlarmExist_i=TRUE AND bAlarmExist_j=TRUE THEN
        	gvl_error.ws_Stasion_In_Error				:= gvl_error.A_Error_station[i_current_alarm].wsStasionInError;
			gvl_error.udi_Station_In_Error 				:= gvl_error.A_Error_station[i_current_alarm].udiStationInError ;
			gvl_error.udi_Station_In_Error_Code 		:= gvl_error.A_Error_description[j_current_alarm].udiStationErrorCode ;
			gvl_error.ws_Station_Error_Description		:= gvl_error.A_Error_description[j_current_alarm].wsStationErrorDescription;
			gvl_error.ws_Station_Error_Description_2 	:= P_ADS_ERR.sStationErrorDescription2;
    	ELSE
		i_current_alarm := 0;
		gvl_error.b_empy_error:=TRUE;
	END_IF
	
END_IF



gvl_error.b_new_system:=bNewSystem;



IF bFirstCycle=TRUE OR b_write=TRUE THEN
	gvl_error.A_Error_station[1].udiStationInError:=1;
	gvl_error.A_Error_station[1].wsStasionInError:="Station1";
	gvl_error.A_Error_description[176].udiStationErrorCode:=311;
	gvl_error.A_Error_description[176].wsStationErrorDescription:="Error176";
	gvl_error.A_Error_description[177].udiStationErrorCode:=18;
	gvl_error.A_Error_description[177].wsStationErrorDescription:="Error177";
	
	FOR k := 2 TO 57 DO
    gvl_error.A_Error_station[k].udiStationInError := 9 + k; // udiStationInError od 11 do 66
    
    wstrStation := WCONCAT("Station", INT_TO_WSTRING(k));
    gvl_error.A_Error_station[k].wsStasionInError := wstrStation;  // Przypisanie wartości WSTRING
	END_FOR
	FOR l := 1 TO 175 DO
    
    wstrStation2 := WCONCAT("Error", INT_TO_WSTRING(l));
    gvl_error.A_Error_description[l].wsStationErrorDescription := wstrStation2;  // Przypisanie wartości WSTRING
	END_FOR
END_IF

IF bFirstCycle=TRUE OR b_write2=TRUE	THEN
	m := 1;  // Inicjalizacja indeksu dla tablicy values
	FOR n := 1 TO 175 DO
    gvl_error.A_Error_description[n].udiStationErrorCode := values[m];  // Przypisanie wartości z tablicy values do A_Error_description
    m := m + 1;  // Przejście do następnej wartości
	END_FOR	

END_IF

IF (previousStationErrorCode <> udiStationErrorCode) AND (udiStationErrorCode <>0)  THEN
	bisAlarmChanged:=TRUE;
END_IF
IF(previousStationErrorCode = udiStationErrorCode) THEN
		bisAlarmChanged:=FALSE;
END_IF
	rTrigError_1(CLK:=bisAlarmChanged);
gvl_error.b_empy_error:=FALSE;

END_PROGRAM

// ---- NotUsedPOU/FB_AssignUserParam.TcPOU
FUNCTION_BLOCK FB_AssignUserParam
VAR
    paramKey, paramValue : STRING(80); // Klucz i wartość parametru
    splitPos            : INT; // Pozycja rozdzielnika między kluczem a wartością
    i                   : INT; // Licznik
    userParams          : ARRAY[1..8] OF STRING(255); // Tablica parametrów
END_VAR

// Iteracja przez parametry
FOR i := 1 TO 8 DO
    splitPos := FIND(userParams[i], ' : '); // Szukamy separatora między kluczem a wartością
    IF splitPos > 0 THEN
        paramKey := LEFT(userParams[i], splitPos - 1); // Klucz
        paramValue := RIGHT(userParams[i], LEN(userParams[i]) - splitPos - 2); // Wartość

        // Sprawdzamy klucz i przypisujemy odpowiednią wartość do struktury użytkownika
        CASE paramKey OF
            'User':	P_UserManagment.user_array[userID].userLogin := paramValue; // Przypisujemy login
            'domain': P_UserManagment.user_array[userID].userGroup := paramValue;
            'autoLogout': P_UserManagment.user_array[userID].autoLogOff := STRING_TO_INT(paramValue); // Konwersja do INT
            'locale': P_UserManagment.user_array[userID].locale := paramValue;
            'timeFormatLocale': P_UserManagment.user_array[userID].timeFormatlocale := paramValue;
            'timeZone': P_UserManagment.user_array[userID].timeZone := paramValue;
            'groups': P_UserManagment.user_array[userID].userGroup := paramValue; // Przypisanie grupy użytkownika
         ELSE
                // Ignorowanie nieznanych kluczy
        END_CASE
    END_IF
END_FOR

END_FUNCTION_BLOCK

// ---- NotUsedPOU/F_ParseKeyValue.TcPOU
FUNCTION F_ParseKeyValue : BOOL
VAR_INPUT
    inputLine : STRING(255);  // Linia do rozdzielenia
END_VAR
VAR_OUTPUT
    key       : STRING(80);   // Klucz
    value     : STRING(80);   // Wartość
END_VAR
VAR
    splitPos  : INT;          // Pozycja separatora ":"
END_VAR

splitPos := FIND(inputLine, ' : ');

IF splitPos > 0 THEN
    key := LEFT(inputLine, splitPos - 1);
    value := RIGHT(inputLine, LEN(inputLine) - splitPos - 2);
    F_ParseKeyValue := TRUE;
ELSE
    F_ParseKeyValue := FALSE;
END_IF

END_FUNCTION

// ---- NotUsedPOU/F_ParseUserString.TcPOU
FUNCTION F_ParseUserString : BOOL
VAR_INPUT
    userString : STRING(1000) :=gvl_his.string_of_properties; // String do rozbicia
END_VAR
VAR
    paramLines : ARRAY[1..100] OF STRING(255);  // Tablica przechowująca linie z parametrami
    lineCount  : INT;                          // Liczba linii w stringu
    paramKey, paramValue : STRING(80);        // Klucz i wartość parametru
    i          : INT;                          // Licznik pętli
END_VAR
VAR_OUTPUT
	user_array :ARRAY[1..100] of string(255);
END_VAR

// Rozdziel string na linie według znaku nowej linii
lineCount := F_SplitStringLines(userString, '\n');

// Iterujemy po liniach stringa i rozdzielamy klucz oraz wartość
FOR i := 1 TO lineCount DO
    IF F_ParseKeyValue(paramLines[i]) THEN
        // Przypisujemy do zmiennych globalnych odpowiednie parametry
        CASE F_ParseKeyValue.key OF
            'User': P_UserManagment.user_array[GVL_USER.currentUser].userLogin := paramValue;
            'domain': P_UserManagment.user_array[GVL_USER.currentUser].userGroup := paramValue;
            'autoLogout': P_UserManagment.user_array[GVL_USER.currentUser].autoLogOff := STRING_TO_INT(paramValue);  // Konwersja na INT
            'locale': P_UserManagment.user_array[GVL_USER.currentUser].locale := paramValue;
            'timeFormatLocale': P_UserManagment.user_array[GVL_USER.currentUser].timeFormatlocale := paramValue;
            'timeZone': P_UserManagment.user_array[GVL_USER.currentUser].timeZone := paramValue;
            'groups': P_UserManagment.user_array[GVL_USER.currentUser].userGroup := paramValue;  // Przypisanie grupy użytkownika
            ELSE
                // Ignorowanie nieznanych kluczy
        END_CASE;
    END_IF;
END_FOR;

F_ParseUserString := TRUE;  // Zwracamy TRUE, jeśli parsowanie się udało

END_FUNCTION

// ---- NotUsedPOU/F_SplitStringLines.TcPOU
FUNCTION F_SplitStringLines : INT
VAR_INPUT
    userString : STRING(1024);  // String do podziału
    separator   : STRING(1);    // Separator (np. '\n')
END_VAR
VAR_OUTPUT
    linesArray  : ARRAY[1..100] OF STRING(255);  // Tablica linii
END_VAR
VAR
    pos         : INT;           // Pozycja separatora
    startPos    : INT;           // Pozycja początku nowej linii
    lineCount   : INT := 0;     // Licznik linii
END_VAR

startPos := 1;

WHILE LEN(userString) > 0 DO
    pos := FIND(userString, separator);
    IF pos > 0 THEN
        linesArray[lineCount + 1] := LEFT(userString, pos - 1);
        userString := RIGHT(userString, LEN(userString) - pos - LEN(separator) + 1);
        lineCount := lineCount + 1;
    ELSE
        linesArray[lineCount + 1] := userString;
        userString := '';
        lineCount := lineCount + 1;
    END_IF
END_WHILE

F_SplitStringLines := lineCount;  // Zwracamy liczbę linii

END_FUNCTION

// ---- NotUsedPOU/P_EvtLog.TcPOU
PROGRAM P_EvtLog
VAR
	alarm : FB_TcAlarm;
	state: INT;
	raise: BOOL;
	clear: BOOL;
END_VAR

CASE state OF
	0:
		alarm.Create(
			eventClass			:= TC_EVENT_CLASSES.NewEventClass, 
			nEventId			:= TC_EVENTS.NewEventClass.Event.nEventId, 
			eSeverity			:= TcEventSeverity.Error, 
			bWithConfirmation	:= FALSE, 
			ipSourceInfo		:= 0);
		state := 10;
		
	10:
		alarm.ipArguments.Clear().AddString('Tekst1').AddString('Tekst2').AddString('Tekst3');
		state := 20;
		
	20:
		IF raise THEN
			alarm.Raise(0);
		END_IF
		IF clear THEN
			alarm.Clear(0, FALSE);
		END_IF
END_CASE

END_PROGRAM

// ---- NotUsedPOU/P_ParseString.TcPOU
PROGRAM P_ParseString
VAR
    result     : BOOL;  // Zmienna pomocnicza do sprawdzenia wyniku parsowania
END_VAR

// Sprawdzenie, czy string z HMI nie jest pusty
IF LEN(gvl_his.string_of_properties) > 0 THEN
    result := F_ParseUserString(gvl_his.string_of_properties);  // Wywołanie funkcji parsującej string

    IF result THEN
        GVL_USER.currentUser := GVL_USER.currentUser + 1;  // Zwiększamy indeks dla następnego użytkownika
        IF GVL_USER.currentUser > 100 THEN
            GVL_USER.currentUser := 1;  // Zawijamy indeks, gdy przekroczymy 100 użytkowników
        END_IF;
    END_IF;
END_IF;

END_PROGRAM

// ---- NotUsedPOU/P_UserDataManagment.TcPOU
PROGRAM P_UserDataManagment
VAR
    inputString : STRING(1000);
	line : STRING(255);          // Linia aktualnie przetwarzana
    key : STRING(80);            // Klucz
    value : STRING(80);          // Wartość
    pos : INT;                   // Pozycja separatora
    index : INT;                 // Indeks w tablicy
    lineCount : INT;             // Liczba linii przetworzonych
    userLineCount : INT;         // Liczba użytkowników przetworzonych
END_VAR

inputString := GVL_USER.string_of_properties;  // Odczytaj string z HMI

lineCount := 0;
userLineCount := 0;
index := 0;

// Rozdziel string na linie
WHILE LEN(inputString) > 0 DO
    pos := FIND(inputString, '\n');
    IF pos > 0 THEN
        line := LEFT(inputString, pos - 1);
        inputString := RIGHT(inputString, LEN(inputString) - pos - 1);
    ELSE
        line := inputString;
        inputString := '';
    END_IF

    // Sprawdź, czy linia zawiera dane użytkownika
    IF FIND(line, 'User:') > 0 THEN
        // Nowy użytkownik
        index := userLineCount;
        userLineCount := userLineCount + 1;
        CONTINUE;
    END_IF

    // Rozdziel linię na klucz i wartość
    pos := FIND(line, ' : ');  // Zakładamy, że separator to " : "
    IF pos > 0 THEN
        key := LEFT(line, pos - 1);
        value := RIGHT(line, LEN(line) - pos - 2);

        // Przypisz wartości do odpowiednich pól w tablicy
		IF	key = 'User' THEN
			GVL_USER.user_array[index].password := value;
			GVL_USER.user_array[index].userLogin := value;
        ELSIF key = 'domain' THEN
            GVL_USER.user_array[index].domain := value;
        ELSIF key = 'enabled' THEN
            GVL_USER.user_array[index].enabled := TRUE;  // Konwersja na BOOL
        ELSIF key = 'autoLogout' THEN
            GVL_USER.user_array[index].autoLogOff := value;  // Konwersja na INT
        ELSIF key = 'locale' THEN
            GVL_USER.user_array[index].locale := value;
        ELSIF key = 'groups' THEN
            GVL_USER.user_array[index].userGroup := value;  // Przypisanie grupy użytkownika
        ELSE
            // Ignorowanie nieznanych kluczy
        END_IF
    END_IF

    lineCount := lineCount + 1;
END_WHILE

END_PROGRAM

// ---- POUs/FB_SaveLineToFile.TcPOU
(****************************************************************************************)
(*							Beckhoff Automation Poland									*)
(*								FB_SaveLineToFile  v2.0									*)
(*									26.06.2014											*)
(*						Blok funkcyjny zapisujacy tekst do pliku						*)
(*______________________________________________________________________________________
	Versions:
		v1.1	05.08.2016	* Przepisana wersja do TwinCat3
		v1.0	17.09.2012	* Podstawowa wersja z TwinCat2
________________________________________________________________________________________*)
FUNCTION_BLOCK FB_SaveLineToFile
VAR_INPUT
	bExecute	: BOOL;			(* Komenda wpisu *)
	AmsNetId	: T_AmsNetId;	(* AMS NET ID obiektu docelowego, gdy lokalnie, to zmienna moze byc pusta *)
	sPath		: STRING; 		(* Sciezka pliku, np  'Hard Disk\'*)
	sName		: STRING; 		(* Nazwa pliku wraz z rozszerzeniem 'LogFile.txt'; *)
	sLine		: STRING;		(* Tresc wpisu *)
END_VAR
VAR_OUTPUT
	bBusy		: BOOL;
	bError		: BOOL;
END_VAR
VAR
	fbFileOpen	: FB_FileOpen;
	ftOpen		: F_TRIG;
	fbFilePuts	: FB_FilePuts;
	ftPuts		: F_TRIG;
	fbFileClose	: FB_FileClose;
	ftClose		: F_TRIG;
END_VAR
VAR // added by the converter: edge detectors and wires of the graphical bodies
    _w1 : BOOL;
END_VAR

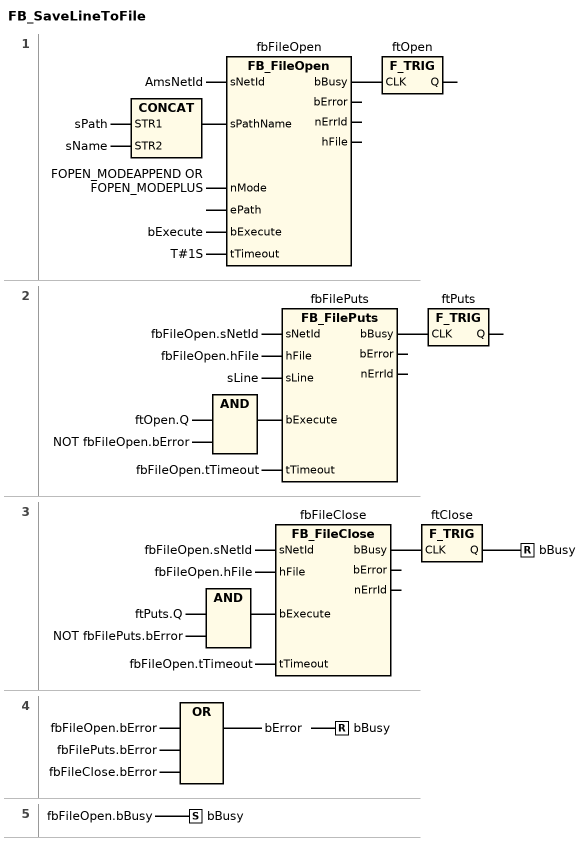
// NETWORK 1
fbFileOpen(
    sNetId := AmsNetId,
    sPathName := CONCAT(STR1 := sPath, STR2 := sName),
    nMode := FOPEN_MODEAPPEND OR FOPEN_MODEPLUS,
    bExecute := bExecute,
    tTimeout := T#1S); // FB_FileOpen
ftOpen(CLK := fbFileOpen.bBusy); // F_TRIG

// NETWORK 2
fbFilePuts(
    sNetId := fbFileOpen.sNetId,
    hFile := fbFileOpen.hFile,
    sLine := sLine,
    bExecute := ftOpen.Q AND (NOT fbFileOpen.bError),
    tTimeout := fbFileOpen.tTimeout); // FB_FilePuts
ftPuts(CLK := fbFilePuts.bBusy); // F_TRIG

// NETWORK 3
fbFileClose(
    sNetId := fbFileOpen.sNetId,
    hFile := fbFileOpen.hFile,
    bExecute := ftPuts.Q AND (NOT fbFilePuts.bError),
    tTimeout := fbFileOpen.tTimeout); // FB_FileClose
ftClose(CLK := fbFileClose.bBusy); // F_TRIG
bBusy R= ftClose.Q;

